KUKA KRL program: MyProgram_164().src

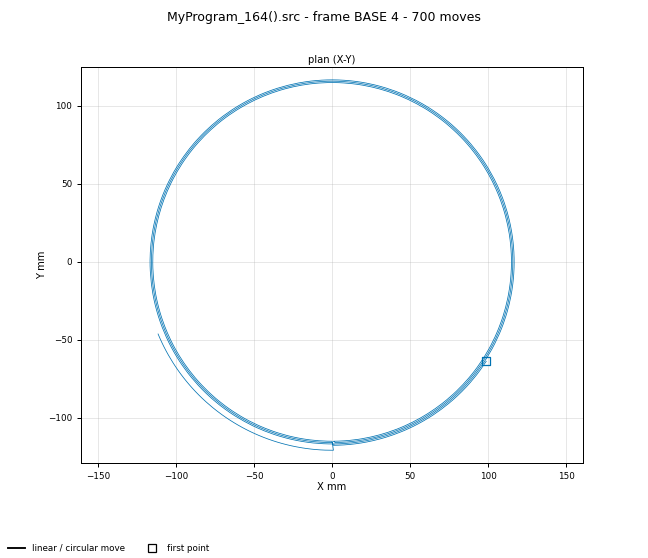
[picture p0: tool path of MyProgram_164().src in frame BASE 4, 700 of 700 moves have a stored position in this frame; points joined in program order, loops and branches not executed]
&ACCESS RVP
&REL 1
&PARAM TEMPLATE = C:\KRC\Roboter\Template\vorgabe
&PARAM EDITMASK = *
DEF MyProgram_164()
; ---- Setting reference (Base) ----
$BASE = BASE_DATA[4]

; --------------------------
; ---- Setting tool (TCP) ----
$TOOL = TOOL_DATA[3]
; --------------------------

$VEL.CP = VEL_APROX_PRINT
Startdeposition()
$VEL.CP = VEL_PRINT
LIN {X 98.7542,Y -63.6993,Z 124,A -36.9555,B 24.954,C -1.5673,E1 25.1338,E2 483.0384} C_DIS
LIN {X 95.0307,Y -69.1319,Z 124,A -40.7241,B 24.956,C -1.5319,E1 25.1276,E2 486.872} C_DIS
LIN {X 92.4043,Y -72.6049,Z 124,A -42.0258,B 24.9541,C -1.565,E1 25.1255,E2 488.0895} C_DIS
LIN {X 88.5317,Y -77.2791,Z 124,A -45.1866,B 24.9551,C -1.5476,E1 25.1198,E2 491.2768} C_DIS
LIN {X 86.1751,Y -79.9009,Z 124,A -47.118,B 24.956,C -1.5331,E1 25.1161,E2 493.234} C_DIS
LIN {X 83.1674,Y -83.0271,Z 124,A -49.5456,B 24.9571,C -1.5131,E1 25.1113,E2 495.6983} C_DIS
LIN {X 80.2255,Y -85.8716,Z 124,A -51.1384,B 24.9563,C -1.5272,E1 25.1081,E2 497.2513} C_DIS
LIN {X 77.3974,Y -88.4284,Z 124,A -52.8872,B 24.9563,C -1.5281,E1 25.1045,E2 498.9912} C_DIS
LIN {X 74.8233,Y -90.6175,Z 124,A -54.4447,B 24.9563,C -1.5286,E1 25.1012,E2 500.5415} C_DIS
LIN {X 69.7732,Y -94.5611,Z 124,A -57.4094,B 24.9562,C -1.5292,E1 25.0947,E2 503.4937} C_DIS
LIN {X 64.9685,Y -97.9241,Z 124,A -60.2141,B 24.9564,C -1.5259,E1 25.0883,E2 506.2966} C_DIS
LIN {X 62.6063,Y -99.4512,Z 124,A -61.8472,B 24.9572,C -1.5109,E1 25.0843,E2 507.9599} C_DIS
LIN {X 58.7888,Y -101.754,Z 124,A -64.5484,B 24.9588,C -1.4824,E1 25.0777,E2 510.7201} C_DIS
LIN {X 55.0039,Y -103.8486,Z 124,A -66.1004,B 24.9576,C -1.5045,E1 25.074,E2 512.2154} C_DIS
LIN {X 51.9264,Y -105.4213,Z 124,A -68.4778,B 24.9595,C -1.4698,E1 25.0679,E2 514.6687} C_DIS
LIN {X 47.367,Y -107.5476,Z 124,A -70.0158,B 24.9574,C -1.5081,E1 25.0642,E2 516.1122} C_DIS
LIN {X 44.6784,Y -108.6919,Z 124,A -71.6622,B 24.9581,C -1.4958,E1 25.0599,E2 517.784} C_DIS
LIN {X 39.1961,Y -110.7866,Z 124,A -74.7628,B 24.9589,C -1.4809,E1 25.0517,E2 520.9132} C_DIS
LIN {X 34.6946,Y -112.2774,Z 124,A -76.7337,B 24.9582,C -1.4937,E1 25.0465,E2 522.85} C_DIS
LIN {X 31.2285,Y -113.2919,Z 124,A -79.3158,B 24.9604,C -1.4543,E1 25.0394,E2 525.5212} C_DIS
LIN {X 26.1754,Y -114.5637,Z 124,A -80.5685,B 24.9572,C -1.5106,E1 25.0363,E2 526.6388} C_DIS
LIN {X 22.2355,Y -115.3928,Z 124,A -82.9862,B 24.9585,C -1.488,E1 25.0296,E2 529.1072} C_DIS
LIN {X 18.6888,Y -116.0221,Z 124,A -84.9192,B 24.959,C -1.4785,E1 25.0242,E2 531.0604} C_DIS
LIN {X 14.9785,Y -116.5572,Z 124,A -86.5895,B 24.9587,C -1.4845,E1 25.0196,E2 532.7153} C_DIS
LIN {X 11.1662,Y -116.9845,Z 124,A -88.5257,B 24.9589,C -1.4804,E1 25.0142,E2 534.6598} C_DIS
LIN {X 7.7029,Y -117.2631,Z 124,A -90.1788,B 24.9589,C -1.4815,E1 25.0096,E2 536.3096} C_DIS
LIN {X 3.8149,Y -117.4539,Z 124,A -92.07,B 24.9589,C -1.4811,E1 25.0043,E2 538.2012} C_DIS
LIN {X 0.8269,Y -117.5118,Z 124,A -92.9024,B 24.9573,C -1.509,E1 25.0022,E2 538.9674} C_DIS
Enddeposition()
LIN {X 0.8269,Y -117.5118,Z 124,A -92.9024,B 24.9573,C -1.509,E1 25.0022,E2 538.9674} C_DIS
Startdeposition()
$VEL.CP = VEL_PRINT
LIN {X 1.3624,Y -116.6412,Z 124,A -92.4871,B 24.9561,C -1.5309,E1 25.0035,E2 538.5001} C_DIS
LIN {X 4.937,Y -116.5432,Z 124,A -90.7988,B 24.9562,C -1.5285,E1 25.0082,E2 536.8181} C_DIS
LIN {X 8.3454,Y -116.3498,Z 124,A -89.0348,B 24.956,C -1.5332,E1 25.0131,E2 535.0436} C_DIS
LIN {X 12.1794,Y -116.0101,Z 124,A -87.2047,B 24.956,C -1.5315,E1 25.0182,E2 533.2187} C_DIS
LIN {X 16.0648,Y -115.5367,Z 124,A -85.3224,B 24.956,C -1.5309,E1 25.0234,E2 531.3393} C_DIS
LIN {X 19.0946,Y -115.0744,Z 124,A -83.8374,B 24.956,C -1.5311,E1 25.0275,E2 529.8554} C_DIS
LIN {X 21.8358,Y -114.5859,Z 124,A -82.4991,B 24.956,C -1.5308,E1 25.0312,E2 528.5191} C_DIS
LIN {X 24.7791,Y -113.9855,Z 124,A -80.9678,B 24.9559,C -1.5347,E1 25.0354,E2 526.9805} C_DIS
LIN {X 33.0953,Y -111.8544,Z 124,A -76.9507,B 24.9562,C -1.5298,E1 25.0462,E2 522.9812} C_DIS
LIN {X 36.0082,Y -110.9509,Z 124,A -75.15,B 24.9552,C -1.5457,E1 25.0511,E2 521.1465} C_DIS
LIN {X 40.8071,Y -109.2778,Z 124,A -72.5586,B 24.9548,C -1.5534,E1 25.0579,E2 518.5422} C_DIS
LIN {X 45.2858,Y -107.4983,Z 124,A -70.3865,B 24.9551,C -1.5477,E1 25.0635,E2 516.3884} C_DIS
LIN {X 47.8668,Y -106.3742,Z 124,A -68.1457,B 24.9526,C -1.5902,E1 25.0694,E2 514.0527} C_DIS
LIN {X 52.9793,Y -103.9226,Z 124,A -66.2695,B 24.9549,C -1.552,E1 25.0739,E2 512.272} C_DIS
LIN {X 58.1058,Y -101.1455,Z 124,A -62.9534,B 24.9533,C -1.5784,E1 25.0821,E2 508.9032} C_DIS
LIN {X 61.3448,Y -99.2159,Z 124,A -61.5325,B 24.9543,C -1.5615,E1 25.0854,E2 507.5266} C_DIS
LIN {X 64.5929,Y -97.1322,Z 124,A -59.0864,B 24.9525,C -1.5914,E1 25.0912,E2 505.0181} C_DIS
LIN {X 68.1356,Y -94.6808,Z 124,A -57.4862,B 24.9537,C -1.5713,E1 25.0947,E2 503.471} C_DIS
LIN {X 73.0483,Y -90.9445,Z 124,A -54.5115,B 24.9535,C -1.5752,E1 25.1013,E2 500.498} C_DIS
LIN {X 75.6279,Y -88.8094,Z 124,A -52.8968,B 24.9534,C -1.5775,E1 25.1047,E2 498.884} C_DIS
LIN {X 78.6353,Y -86.1583,Z 124,A -50.8669,B 24.9529,C -1.585,E1 25.109,E2 496.8446} C_DIS
LIN {X 82.5495,Y -82.4176,Z 124,A -48.2216,B 24.9526,C -1.5908,E1 25.1143,E2 494.1967} C_DIS
LIN {X 84.4942,Y -80.4234,Z 124,A -46.9043,B 24.9526,C -1.5918,E1 25.1168,E2 492.8826} C_DIS
LIN {X 86.8418,Y -77.8794,Z 124,A -45.2097,B 24.9523,C -1.5959,E1 25.12,E2 491.1858} C_DIS
LIN {X 90.3208,Y -73.8178,Z 124,A -42.6097,B 24.9519,C -1.6016,E1 25.1247,E2 488.5843} C_DIS
LIN {X 91.9446,Y -71.7869,Z 124,A -41.019,B 24.9508,C -1.62,E1 25.1275,E2 486.9576} C_DIS
LIN {X 95.3627,Y -67.1797,Z 124,A -38.1108,B 24.9501,C -1.6322,E1 25.1322,E2 484.0347} C_DIS
LIN {X 97.3923,Y -64.1983,Z 124,A -36.8892,B 24.9514,C -1.6108,E1 25.134,E2 482.8696} C_DIS
LIN {X 99.3478,Y -61.132,Z 124,A -35.1139,B 24.9511,C -1.6154,E1 25.1367,E2 481.0925} C_DIS
LIN {X 102.5848,Y -55.5254,Z 124,A -31.853,B 24.9503,C -1.6287,E1 25.1412,E2 477.8173} C_DIS
LIN {X 104.3109,Y -52.2123,Z 124,A -30.2141,B 24.9505,C -1.6248,E1 25.1433,E2 476.1963} C_DIS
LIN {X 107.2037,Y -45.9841,Z 124,A -26.5839,B 24.9491,C -1.6474,E1 25.1475,E2 472.5325} C_DIS
LIN {X 108.4916,Y -42.8522,Z 124,A -25.1108,B 24.9494,C -1.6434,E1 25.149,E2 471.0768} C_DIS
LIN {X 109.6343,Y -39.8375,Z 124,A -22.6264,B 24.9463,C -1.6921,E1 25.1515,E2 468.4916} C_DIS
LIN {X 111.3881,Y -34.6323,Z 124,A -20.7918,B 24.9484,C -1.6587,E1 25.153,E2 466.7461} C_DIS
LIN {X 112.2363,Y -31.7759,Z 124,A -18.7125,B 24.9463,C -1.6932,E1 25.1546,E2 464.5973} C_DIS
LIN {X 113.3809,Y -27.414,Z 124,A -17.6096,B 24.9492,C -1.6466,E1 25.1553,E2 463.6107} C_DIS
LIN {X 114.5448,Y -22.0493,Z 124,A -14.4678,B 24.9473,C -1.6766,E1 25.1572,E2 460.4164} C_DIS
LIN {X 115.1793,Y -18.4619,Z 124,A -12.6055,B 24.9467,C -1.686,E1 25.158,E2 458.5431} C_DIS
LIN {X 115.7491,Y -14.461,Z 124,A -10.6706,B 24.9465,C -1.69,E1 25.1587,E2 456.61} C_DIS
LIN {X 116.1418,Y -10.8535,Z 124,A -8.9547,B 24.9463,C -1.6927,E1 25.1592,E2 454.898} C_DIS
LIN {X 116.3878,Y -7.7827,Z 124,A -7.4105,B 24.9459,C -1.6991,E1 25.1595,E2 453.3478} C_DIS
LIN {X 116.5865,Y -3.7859,Z 124,A -5.5405,B 24.9458,C -1.7009,E1 25.1597,E2 451.4846} C_DIS
LIN {X 116.6446,Y -0.9225,Z 124,A -4.0905,B 24.9454,C -1.7076,E1 25.1597,E2 450.0275} C_DIS
LIN {X 116.6233,Y 2.4022,Z 124,A -2.3642,B 24.9447,C -1.7174,E1 25.1597,E2 448.2884} C_DIS
LIN {X 116.4751,Y 6.3448,Z 124,A -0.61,B 24.9449,C -1.7149,E1 25.1595,E2 446.5506} C_DIS
LIN {X 116.2723,Y 9.3509,Z 124,A 0.8728,B 24.9446,C -1.7198,E1 25.1592,E2 445.0649} C_DIS
LIN {X 115.9636,Y 12.6238,Z 124,A 2.6543,B 24.9437,C -1.733,E1 25.1587,E2 443.2628} C_DIS
LIN {X 115.5191,Y 16.1886,Z 124,A 4.2881,B 24.9437,C -1.7324,E1 25.1581,E2 441.6401} C_DIS
LIN {X 114.9628,Y 19.7618,Z 124,A 6.0877,B 24.9433,C -1.7392,E1 25.1573,E2 439.8351} C_DIS
LIN {X 114.2684,Y 23.44,Z 124,A 7.9174,B 24.943,C -1.7446,E1 25.1563,E2 438.0034} C_DIS
LIN {X 113.3834,Y 27.4035,Z 124,A 9.6005,B 24.9435,C -1.7359,E1 25.1552,E2 436.3505} C_DIS
LIN {X 112.2328,Y 31.788,Z 124,A 12.1154,B 24.9422,C -1.7566,E1 25.1534,E2 433.8013} C_DIS
LIN {X 110.4058,Y 37.6486,Z 124,A 15.0322,B 24.9419,C -1.761,E1 25.1509,E2 430.8906} C_DIS
LIN {X 109.1594,Y 41.1212,Z 124,A 16.9719,B 24.9411,C -1.7725,E1 25.149,E2 428.9346} C_DIS
LIN {X 107.5453,Y 45.1743,Z 124,A 18.989,B 24.9411,C -1.7728,E1 25.1469,E2 426.9279} C_DIS
LIN {X 106.1515,Y 48.3609,Z 124,A 20.7337,B 24.9407,C -1.7795,E1 25.1449,E2 425.177} C_DIS
LIN {X 103.7325,Y 53.3512,Z 124,A 23.4235,B 24.9402,C -1.7856,E1 25.1416,E2 422.4872} C_DIS
LIN {X 100.1461,Y 59.8142,Z 124,A 27.1032,B 24.9394,C -1.7978,E1 25.1365,E2 418.7979} C_DIS
LIN {X 98.2857,Y 62.8224,Z 124,A 28.6878,B 24.9396,C -1.7951,E1 25.1342,E2 417.2275} C_DIS
LIN {X 96.7431,Y 65.1731,Z 124,A 30.6198,B 24.9376,C -1.8249,E1 25.1311,E2 415.2348} C_DIS
LIN {X 94.4395,Y 68.4702,Z 124,A 32.0919,B 24.9389,C -1.806,E1 25.1288,E2 413.8145} C_DIS
LIN {X 92.4871,Y 71.0834,Z 124,A 33.6422,B 24.9388,C -1.8075,E1 25.1261,E2 412.2679} C_DIS
LIN {X 89.196,Y 75.1741,Z 124,A 36.3243,B 24.938,C -1.8185,E1 25.1214,E2 409.5723} C_DIS
LIN {X 86.7479,Y 77.9843,Z 124,A 38.0837,B 24.938,C -1.8194,E1 25.1181,E2 407.8187} C_DIS
LIN {X 84.1411,Y 80.7899,Z 124,A 39.925,B 24.9378,C -1.8217,E1 25.1146,E2 405.9799} C_DIS
LIN {X 81.95,Y 83.0114,Z 124,A 41.4369,B 24.9376,C -1.8241,E1 25.1116,E2 404.4688} C_DIS
LIN {X 79.2815,Y 85.5655,Z 124,A 43.304,B 24.9372,C -1.8303,E1 25.1078,E2 402.5947} C_DIS
LIN {X 76.7637,Y 87.8296,Z 124,A 44.9058,B 24.9372,C -1.8308,E1 25.1045,E2 400.998} C_DIS
LIN {X 74.5063,Y 89.7525,Z 124,A 46.9912,B 24.9349,C -1.863,E1 25.0999,E2 398.8446} C_DIS
LIN {X 70.9944,Y 92.5557,Z 124,A 48.5591,B 24.9367,C -1.8372,E1 25.0965,E2 397.3434} C_DIS
LIN {X 67.7868,Y 94.9297,Z 124,A 50.3301,B 24.9371,C -1.832,E1 25.0926,E2 395.5911} C_DIS
LIN {X 64.3975,Y 97.261,Z 124,A 52.5478,B 24.9362,C -1.8444,E1 25.0874,E2 393.3515} C_DIS
LIN {X 61.3344,Y 99.2224,Z 124,A 54.4921,B 24.9355,C -1.8544,E1 25.0828,E2 391.3897} C_DIS
LIN {X 57.7899,Y 101.327,Z 124,A 56.1965,B 24.9364,C -1.8427,E1 25.0787,E2 389.7182} C_DIS
LIN {X 53.6383,Y 103.5858,Z 124,A 58.7779,B 24.9353,C -1.8577,E1 25.0723,E2 387.1086} C_DIS
LIN {X 47.1433,Y 106.6983,Z 124,A 62.2251,B 24.9353,C -1.8578,E1 25.0636,E2 383.6701} C_DIS
LIN {X 43.3275,Y 108.3047,Z 124,A 64.6027,B 24.9341,C -1.8756,E1 25.0574,E2 381.2557} C_DIS
LIN {X 40.2198,Y 109.4949,Z 124,A 65.8533,B 24.9352,C -1.8597,E1 25.0542,E2 380.0454} C_DIS
LIN {X 36.9579,Y 110.6387,Z 124,A 67.5149,B 24.9352,C -1.8595,E1 25.0498,E2 378.3875} C_DIS
LIN {X 34.4288,Y 111.4512,Z 124,A 69.1235,B 24.9341,C -1.8743,E1 25.0455,E2 376.7468} C_DIS
LIN {X 30.1108,Y 112.6949,Z 124,A 71.3904,B 24.9339,C -1.8785,E1 25.0393,E2 374.4737} C_DIS
LIN {X 26.8729,Y 113.5118,Z 124,A 72.7814,B 24.9346,C -1.8681,E1 25.0356,E2 373.1092} C_DIS
LIN {X 21.9765,Y 114.5588,Z 124,A 75.4902,B 24.9337,C -1.8805,E1 25.0281,E2 370.3744} C_DIS
LIN {X 18.6584,Y 115.1473,Z 124,A 76.9039,B 24.9344,C -1.8702,E1 25.0243,E2 368.9866} C_DIS
LIN {X 15.0241,Y 115.6761,Z 124,A 78.5845,B 24.9348,C -1.8652,E1 25.0197,E2 367.3193} C_DIS
LIN {X 11.6126,Y 116.0695,Z 124,A 80.3473,B 24.9345,C -1.8688,E1 25.0148,E2 365.5491} C_DIS
LIN {X 7.9248,Y 116.3782,Z 124,A 82.1279,B 24.9346,C -1.8672,E1 25.0098,E2 363.7731} C_DIS
LIN {X 3.8833,Y 116.5835,Z 124,A 84.1046,B 24.9346,C -1.8666,E1 25.0043,E2 361.7984} C_DIS
LIN {X 0.3729,Y 116.6476,Z 124,A 85.8948,B 24.9346,C -1.8692,E1 24.9993,E2 360.0022} C_DIS
LIN {X -3.3094,Y 116.6011,Z 124,A 87.5792,B 24.9349,C -1.8633,E1 24.9946,E2 358.3318} C_DIS
LIN {X -6.5798,Y 116.4621,Z 124,A 89.2341,B 24.9349,C -1.8648,E1 24.99,E2 356.6728} C_DIS
LIN {X -10.4984,Y 116.1745,Z 124,A 91.1377,B 24.9349,C -1.8628,E1 24.9847,E2 354.7733} C_DIS
LIN {X -13.5851,Y 115.8539,Z 124,A 92.7068,B 24.9349,C -1.8639,E1 24.9804,E2 353.2005} C_DIS
LIN {X -16.8387,Y 115.4268,Z 124,A 94.5371,B 24.9343,C -1.8724,E1 24.9753,E2 351.3486} C_DIS
LIN {X -21.7106,Y 114.61,Z 124,A 96.7704,B 24.935,C -1.8621,E1 24.9692,E2 349.1374} C_DIS
LIN {X -28.2657,Y 113.1728,Z 124,A 100.1287,B 24.935,C -1.8617,E1 24.96,E2 345.7757} C_DIS
LIN {X -34.9527,Y 111.2887,Z 124,A 103.5513,B 24.9353,C -1.8583,E1 24.9509,E2 342.3555} C_DIS
LIN {X -38.7551,Y 110.0216,Z 124,A 105.4456,B 24.9357,C -1.8527,E1 24.9459,E2 340.4709} C_DIS
LIN {X -43.2758,Y 108.3252,Z 124,A 107.8946,B 24.9357,C -1.8527,E1 24.9395,E2 338.0165} C_DIS
LIN {X -46.5236,Y 106.9685,Z 124,A 109.4387,B 24.9364,C -1.8424,E1 24.9356,E2 336.4935} C_DIS
LIN {X -51.4199,Y 104.7037,Z 124,A 112.2036,B 24.9364,C -1.8431,E1 24.9286,E2 333.72} C_DIS
LIN {X -54.3698,Y 103.2018,Z 124,A 113.8261,B 24.9365,C -1.8403,E1 24.9245,E2 332.0998} C_DIS
LIN {X -57.27,Y 101.6221,Z 124,A 115.4265,B 24.9368,C -1.8365,E1 24.9206,E2 330.5038} C_DIS
LIN {X -60.9655,Y 99.449,Z 124,A 118.0379,B 24.9356,C -1.8541,E1 24.9143,E2 327.8426} C_DIS
LIN {X -64.0825,Y 97.4687,Z 124,A 119.3881,B 24.9372,C -1.8309,E1 24.9112,E2 326.5431} C_DIS
LIN {X -69.7578,Y 93.4916,Z 124,A 123.3224,B 24.9361,C -1.8462,E1 24.9022,E2 322.5585} C_DIS
LIN {X -72.9301,Y 91.0403,Z 124,A 124.8934,B 24.9376,C -1.8251,E1 24.8989,E2 321.0321} C_DIS
LIN {X -77.1018,Y 87.5343,Z 124,A 127.5382,B 24.9381,C -1.8177,E1 24.8933,E2 318.3945} C_DIS
LIN {X -79.6573,Y 85.2146,Z 124,A 129.1643,B 24.9385,C -1.8108,E1 24.89,E2 316.7782} C_DIS
LIN {X -81.473,Y 83.4824,Z 124,A 130.4942,B 24.9385,C -1.8119,E1 24.8873,E2 315.4402} C_DIS
LIN {X -83.8363,Y 81.1062,Z 124,A 132.2471,B 24.9385,C -1.8123,E1 24.8838,E2 313.6788} C_DIS
LIN {X -86.6399,Y 78.1049,Z 124,A 134.1116,B 24.9392,C -1.8008,E1 24.8804,E2 311.8335} C_DIS
LIN {X -88.5148,Y 75.9738,Z 124,A 135.6705,B 24.939,C -1.8041,E1 24.8775,E2 310.2597} C_DIS
LIN {X -91.269,Y 72.6417,Z 124,A 137.668,B 24.9397,C -1.7932,E1 24.874,E2 308.2789} C_DIS
LIN {X -95.079,Y 67.5775,Z 124,A 141.0042,B 24.9397,C -1.7939,E1 24.8685,E2 304.9249} C_DIS
LIN {X -98.2141,Y 62.9341,Z 124,A 143.5663,B 24.9407,C -1.7783,E1 24.8645,E2 302.3872} C_DIS
LIN {X -99.5689,Y 60.7682,Z 124,A 145.2412,B 24.9398,C -1.792,E1 24.8621,E2 300.6708} C_DIS
LIN {X -101.4314,Y 57.6082,Z 124,A 147.1001,B 24.94,C -1.7891,E1 24.8595,E2 298.8092} C_DIS
LIN {X -103.2054,Y 54.363,Z 124,A 148.3584,B 24.9419,C -1.7606,E1 24.8579,E2 297.6121} C_DIS
LIN {X -104.4149,Y 52.0025,Z 124,A 149.7102,B 24.942,C -1.7587,E1 24.8562,E2 296.2576} C_DIS
LIN {X -105.6333,Y 49.481,Z 124,A 151.1826,B 24.942,C -1.7586,E1 24.8544,E2 294.7776} C_DIS
LIN {X -107.0948,Y 46.2339,Z 124,A 152.9845,B 24.9422,C -1.7554,E1 24.8524,E2 292.9734} C_DIS
LIN {X -108.5301,Y 42.7541,Z 124,A 154.8745,B 24.9425,C -1.7514,E1 24.8504,E2 291.0824} C_DIS
LIN {X -110.0165,Y 38.7696,Z 124,A 156.8052,B 24.9434,C -1.7383,E1 24.8486,E2 289.172} C_DIS
LIN {X -110.9839,Y 35.9064,Z 124,A 158.3608,B 24.9434,C -1.7365,E1 24.8472,E2 287.6116} C_DIS
LIN {X -112.0389,Y 32.4724,Z 124,A 160.4445,B 24.943,C -1.744,E1 24.8456,E2 285.4981} C_DIS
LIN {X -113.2143,Y 28.0967,Z 124,A 162.2202,B 24.9447,C -1.7184,E1 24.8444,E2 283.7731} C_DIS
LIN {X -114.1826,Y 23.8578,Z 124,A 164.4125,B 24.945,C -1.7138,E1 24.843,E2 281.5788} C_DIS
LIN {X -114.6949,Y 21.2641,Z 124,A 165.9136,B 24.9447,C -1.7179,E1 24.8422,E2 280.0591} C_DIS
LIN {X -115.3693,Y 17.2328,Z 124,A 168.0274,B 24.9448,C -1.7158,E1 24.8413,E2 277.9379} C_DIS
LIN {X -116.0541,Y 11.7593,Z 124,A 170.6852,B 24.9455,C -1.7048,E1 24.8405,E2 275.2902} C_DIS
LIN {X -116.4878,Y 6.1072,Z 124,A 173.6084,B 24.9457,C -1.7014,E1 24.8399,E2 272.3575} C_DIS
LIN {X -116.6433,Y 1.1077,Z 124,A 175.8997,B 24.9467,C -1.6866,E1 24.8398,E2 270.0878} C_DIS
LIN {X -116.6229,Y -2.4209,Z 124,A 177.5955,B 24.9471,C -1.6794,E1 24.8398,E2 268.3989} C_DIS
LIN {X -116.498,Y -5.9283,Z 124,A 179.4939,B 24.9471,C -1.681,E1 24.8401,E2 266.4853} C_DIS
LIN {X -115.7697,Y -14.3023,Z 124,A -176.2617,B 24.9476,C -1.6724,E1 24.8413,E2 262.236} C_DIS
LIN {X -114.8264,Y -20.5328,Z 124,A -172.8352,B 24.9473,C -1.6763,E1 24.8428,E2 258.7797} C_DIS
LIN {X -114.039,Y -24.5339,Z 124,A -171.3242,B 24.949,C -1.6496,E1 24.8437,E2 257.3235} C_DIS
LIN {X -113.287,Y -27.7986,Z 124,A -169.2783,B 24.9483,C -1.6611,E1 24.845,E2 255.2383} C_DIS
LIN {X -112.3749,Y -31.2866,Z 124,A -167.8442,B 24.9495,C -1.6416,E1 24.8461,E2 253.8423} C_DIS
LIN {X -111.3302,Y -34.8191,Z 124,A -166.0795,B 24.95,C -1.6342,E1 24.8475,E2 252.085} C_DIS
LIN {X -110.1425,Y -38.4105,Z 124,A -164.1882,B 24.9502,C -1.63,E1 24.8492,E2 250.193} C_DIS
LIN {X -108.833,Y -41.983,Z 124,A -162.2156,B 24.9502,C -1.6287,E1 24.8511,E2 248.2124} C_DIS
LIN {X -106.2298,Y -48.1873,Z 124,A -158.9883,B 24.9511,C -1.6159,E1 24.8547,E2 244.9978} C_DIS
LIN {X -104.7752,Y -51.2758,Z 124,A -157.21,B 24.9511,C -1.6153,E1 24.8569,E2 243.2112} C_DIS
LIN {X -103.1018,Y -54.5597,Z 124,A -155.5677,B 24.9518,C -1.6033,E1 24.8589,E2 241.5888} C_DIS
LIN {X -101.3249,Y -57.7935,Z 124,A -153.6752,B 24.9519,C -1.6017,E1 24.8615,E2 239.6903} C_DIS
LIN {X -99.7723,Y -60.4336,Z 124,A -151.8165,B 24.9513,C -1.6125,E1 24.8643,E2 237.7961} C_DIS
LIN {X -98.0488,Y -63.1915,Z 124,A -150.5899,B 24.9525,C -1.5927,E1 24.8661,E2 236.6105} C_DIS
LIN {X -96.1967,Y -65.9801,Z 124,A -148.8284,B 24.9525,C -1.5934,E1 24.8688,E2 234.8387} C_DIS
LIN {X -94.1441,Y -68.8737,Z 124,A -147.1468,B 24.9528,C -1.5865,E1 24.8716,E2 233.1653} C_DIS
LIN {X -92.5609,Y -70.9876,Z 124,A -145.3656,B 24.9518,C -1.6038,E1 24.8747,E2 231.3344} C_DIS
LIN {X -90.116,Y -74.0689,Z 124,A -144.0026,B 24.9535,C -1.575,E1 24.877,E2 230.0336} C_DIS
LIN {X -85.6839,Y -79.1525,Z 124,A -140.4608,B 24.9534,C -1.5771,E1 24.8836,E2 226.471} C_DIS
LIN {X -83.006,Y -81.9554,Z 124,A -138.6761,B 24.9539,C -1.5679,E1 24.887,E2 224.7006} C_DIS
LIN {X -81.0293,Y -83.9104,Z 124,A -137.2764,B 24.954,C -1.5664,E1 24.8898,E2 223.2984} C_DIS
LIN {X -78.1281,Y -86.6191,Z 124,A -135.516,B 24.9547,C -1.5544,E1 24.8934,E2 221.5595} C_DIS
LIN {X -75.9544,Y -88.53,Z 124,A -133.151,B 24.9525,C -1.5922,E1 24.8986,E2 219.0954} C_DIS
LIN {X -71.9938,Y -91.7811,Z 124,A -131.2622,B 24.9544,C -1.5603,E1 24.9026,E2 217.2754} C_DIS
LIN {X -68.7307,Y -94.2488,Z 124,A -129.2623,B 24.9546,C -1.5564,E1 24.9071,E2 215.2778} C_DIS
LIN {X -65.5885,Y -96.4618,Z 124,A -127.425,B 24.9549,C -1.551,E1 24.9113,E2 213.4469} C_DIS
LIN {X -62.3223,Y -98.6053,Z 124,A -125.4267,B 24.9549,C -1.5514,E1 24.916,E2 211.4413} C_DIS
LIN {X -56.3389,Y -102.142,Z 124,A -122.2059,B 24.9557,C -1.5381,E1 24.9237,E2 208.2425} C_DIS
LIN {X -50.9398,Y -104.9383,Z 124,A -119.0798,B 24.9555,C -1.5403,E1 24.9315,E2 205.1027} C_DIS
LIN {X -47.9027,Y -106.358,Z 124,A -117.4982,B 24.9558,C -1.5356,E1 24.9355,E2 203.5284} C_DIS
LIN {X -43.039,Y -108.4182,Z 124,A -114.8225,B 24.9558,C -1.5365,E1 24.9424,E2 200.8447} C_DIS
LIN {X -39.7365,Y -109.6712,Z 124,A -113.1495,B 24.956,C -1.5321,E1 24.9468,E2 199.1785} C_DIS
LIN {X -37.2124,Y -110.5528,Z 124,A -111.5694,B 24.9554,C -1.5428,E1 24.9511,E2 197.5699} C_DIS
LIN {X -33.5458,Y -111.7207,Z 124,A -109.5834,B 24.9552,C -1.5457,E1 24.9564,E2 195.5738} C_DIS
LIN {X -29.0685,Y -112.9678,Z 124,A -107.6872,B 24.9563,C -1.5271,E1 24.9614,E2 193.7188} C_DIS
LIN {X -26.3497,Y -113.6327,Z 124,A -106.2072,B 24.9561,C -1.5311,E1 24.9654,E2 192.2275} C_DIS
LIN {X -22.5124,Y -114.4557,Z 124,A -104.2673,B 24.9561,C -1.5308,E1 24.9708,E2 190.286} C_DIS
LIN {X -19.1502,Y -115.0651,Z 124,A -102.6503,B 24.9563,C -1.5275,E1 24.9752,E2 188.6753} C_DIS
LIN {X -15.2619,Y -115.6453,Z 124,A -100.8004,B 24.9565,C -1.5234,E1 24.9803,E2 186.8336} C_DIS
LIN {X -12.0498,Y -116.0237,Z 124,A -99.1028,B 24.9563,C -1.5281,E1 24.985,E2 185.1238} C_DIS
LIN {X -8.1648,Y -116.362,Z 124,A -97.2841,B 24.9565,C -1.5237,E1 24.9901,E2 183.3147} C_DIS
LIN {X -5.6175,Y -116.5133,Z 124,A -95.9012,B 24.9562,C -1.5296,E1 24.994,E2 181.9175} C_DIS
LIN {X -2.1692,Y -116.6276,Z 124,A -94.2855,B 24.9564,C -1.5263,E1 24.9984,E2 180.3094} C_DIS
LIN {X 0.8245,Y -116.6427,Z 124,A -93.3941,B 24.9578,C -1.5006,E1 25.0008,E2 179.4789} C_DIS
Enddeposition()
LIN {X 0.8245,Y -116.6427,Z 124,A -93.3941,B 24.9578,C -1.5006,E1 25.0008,E2 179.4789} C_DIS
Startdeposition()
$VEL.CP = VEL_PRINT
LIN {X -0.0422,Y -115.7818,Z 124,A -94.1118,B 24.9577,C -1.5029,E1 24.9988,E2 180.1911} C_DIS
LIN {X -3.596,Y -115.724,Z 124,A -95.6773,B 24.9572,C -1.5112,E1 24.9945,E2 181.7372} C_DIS
LIN {X -6.6918,Y -115.5867,Z 124,A -97.2377,B 24.9572,C -1.5099,E1 24.9901,E2 183.301} C_DIS
LIN {X -10.2839,Y -115.3228,Z 124,A -99.0208,B 24.9572,C -1.5099,E1 24.9851,E2 185.0848} C_DIS
LIN {X -12.8754,Y -115.0632,Z 124,A -100.4846,B 24.9577,C -1.5024,E1 24.981,E2 186.5674} C_DIS
LIN {X -16.5458,Y -114.5918,Z 124,A -102.2637,B 24.9576,C -1.5051,E1 24.9761,E2 188.3415} C_DIS
LIN {X -19.9681,Y -114.0462,Z 124,A -103.9919,B 24.9576,C -1.5051,E1 24.9713,E2 190.0715} C_DIS
LIN {X -22.9478,Y -113.4834,Z 124,A -105.2898,B 24.957,C -1.5144,E1 24.9678,E2 191.3484} C_DIS
LIN {X -25.2419,Y -112.9963,Z 124,A -106.8395,B 24.958,C -1.4981,E1 24.9635,E2 192.9389} C_DIS
LIN {X -29.5057,Y -111.9592,Z 124,A -108.727,B 24.9572,C -1.5116,E1 24.9585,E2 194.797} C_DIS
LIN {X -32.3563,Y -111.1683,Z 124,A -110.3907,B 24.9576,C -1.504,E1 24.954,E2 196.4815} C_DIS
LIN {X -36.0487,Y -110.0257,Z 124,A -112.272,B 24.9575,C -1.5068,E1 24.949,E2 198.3594} C_DIS
LIN {X -39.2828,Y -108.9128,Z 124,A -113.6426,B 24.9566,C -1.5221,E1 24.9454,E2 199.6963} C_DIS
LIN {X -41.3773,Y -108.1344,Z 124,A -114.9491,B 24.957,C -1.5145,E1 24.942,E2 201.0236} C_DIS
LIN {X -45.0569,Y -106.653,Z 124,A -116.9742,B 24.957,C -1.5139,E1 24.9367,E2 203.0547} C_DIS
LIN {X -48.7207,Y -105.0299,Z 124,A -118.8384,B 24.9566,C -1.5212,E1 24.932,E2 204.9061} C_DIS
LIN {X -52.5733,Y -103.1554,Z 124,A -121.0937,B 24.9568,C -1.5181,E1 24.9263,E2 207.1747} C_DIS
LIN {X -56.0252,Y -101.3232,Z 124,A -122.9632,B 24.9565,C -1.5234,E1 24.9218,E2 209.0369} C_DIS
LIN {X -59.6868,Y -99.2105,Z 124,A -124.9633,B 24.9561,C -1.5304,E1 24.917,E2 211.0265} C_DIS
LIN {X -62.4196,Y -97.513,Z 124,A -126.6449,B 24.9561,C -1.5291,E1 24.913,E2 212.7165} C_DIS
LIN {X -65.318,Y -95.5969,Z 124,A -128.5187,B 24.9564,C -1.5254,E1 24.9086,E2 214.6054} C_DIS
LIN {X -68.5163,Y -93.3301,Z 124,A -130.4248,B 24.9561,C -1.5301,E1 24.9043,E2 216.5068} C_DIS
LIN {X -71.972,Y -90.6921,Z 124,A -133.4816,B 24.958,C -1.4966,E1 24.8974,E2 219.6546} C_DIS
LIN {X -76.6836,Y -86.7472,Z 124,A -135.4828,B 24.9552,C -1.5455,E1 24.8934,E2 221.5474} C_DIS
LIN {X -79.6326,Y -84.0464,Z 124,A -137.5238,B 24.9552,C -1.547,E1 24.8892,E2 223.5931} C_DIS
LIN {X -82.15,Y -81.587,Z 124,A -139.299,B 24.955,C -1.5493,E1 24.8857,E2 225.3703} C_DIS
LIN {X -84.9958,Y -78.6187,Z 124,A -141.8744,B 24.9561,C -1.5316,E1 24.8807,E2 227.9991} C_DIS
LIN {X -87.7517,Y -75.5311,Z 124,A -143.2769,B 24.9542,C -1.5628,E1 24.8782,E2 229.3336} C_DIS
LIN {X -89.6499,Y -73.2672,Z 124,A -145.0165,B 24.9547,C -1.5548,E1 24.8751,E2 231.1002} C_DIS
LIN {X -92.1975,Y -70.0352,Z 124,A -146.9588,B 24.9542,C -1.5637,E1 24.8718,E2 233.0307} C_DIS
LIN {X -93.9354,Y -67.686,Z 124,A -148.2208,B 24.9535,C -1.5749,E1 24.8697,E2 234.2722} C_DIS
LIN {X -95.2585,Y -65.8095,Z 124,A -149.6237,B 24.954,C -1.5668,E1 24.8675,E2 235.7011} C_DIS
LIN {X -97.1533,Y -62.98,Z 124,A -151.0497,B 24.9531,C -1.5818,E1 24.8653,E2 237.0986} C_DIS
LIN {X -98.2787,Y -61.2069,Z 124,A -152.3631,B 24.9536,C -1.5734,E1 24.8633,E2 238.4389} C_DIS
LIN {X -100.3558,Y -57.738,Z 124,A -154.3082,B 24.9532,C -1.581,E1 24.8606,E2 240.3758} C_DIS
LIN {X -102.4039,Y -54.0224,Z 124,A -156.2743,B 24.9525,C -1.5923,E1 24.858,E2 242.3254} C_DIS
LIN {X -103.7001,Y -51.4904,Z 124,A -157.7403,B 24.9525,C -1.5938,E1 24.8561,E2 243.7956} C_DIS
LIN {X -105.233,Y -48.2845,Z 124,A -159.7043,B 24.9526,C -1.5905,E1 24.8538,E2 245.7782} C_DIS
LIN {X -106.4373,Y -45.5687,Z 124,A -161.292,B 24.9526,C -1.59,E1 24.852,E2 247.3759} C_DIS
LIN {X -108.2244,Y -41.1397,Z 124,A -163.3931,B 24.9516,C -1.6076,E1 24.8499,E2 249.4468} C_DIS
LIN {X -109.4716,Y -37.7012,Z 124,A -165.1706,B 24.9512,C -1.6143,E1 24.8483,E2 251.2184} C_DIS
LIN {X -110.3851,Y -34.9364,Z 124,A -166.7501,B 24.9512,C -1.6131,E1 24.8469,E2 252.8099} C_DIS
LIN {X -111.5631,Y -30.9683,Z 124,A -168.8202,B 24.9509,C -1.6185,E1 24.8453,E2 254.879} C_DIS
LIN {X -112.5089,Y -27.3264,Z 124,A -170.632,B 24.9504,C -1.6264,E1 24.8441,E2 256.6827} C_DIS
LIN {X -113.3734,Y -23.4839,Z 124,A -172.648,B 24.9502,C -1.6298,E1 24.8429,E2 258.7025} C_DIS
LIN {X -114.4548,Y -17.4674,Z 124,A -175.68,B 24.9497,C -1.6391,E1 24.8414,E2 261.7302} C_DIS
LIN {X -114.9715,Y -13.6583,Z 124,A -177.8676,B 24.95,C -1.6338,E1 24.8407,E2 263.9436} C_DIS
LIN {X -115.5236,Y -7.6987,Z 124,A 179.9064,B 24.9476,C -1.6729,E1 24.8402,E2 266.0897} C_DIS
LIN {X -115.735,Y -3.2375,Z 124,A 177.1302,B 24.9485,C -1.6573,E1 24.8398,E2 268.9198} C_DIS
LIN {X -115.778,Y 0.7173,Z 124,A 174.8092,B 24.949,C -1.6491,E1 24.8398,E2 271.2742} C_DIS
LIN {X -115.6929,Y 4.5094,Z 124,A 172.4654,B 24.9498,C -1.6369,E1 24.8401,E2 273.6614} C_DIS
LIN {X -115.3256,Y 10.253,Z 124,A 170.1633,B 24.9479,C -1.6677,E1 24.8406,E2 275.9038} C_DIS
LIN {X -114.9957,Y 13.4524,Z 124,A 168.8931,B 24.9467,C -1.6857,E1 24.841,E2 277.1387} C_DIS
LIN {X -114.4868,Y 17.2605,Z 124,A 166.91,B 24.9466,C -1.6886,E1 24.8418,E2 279.1267} C_DIS
LIN {X -113.8218,Y 21.2142,Z 124,A 164.8586,B 24.9463,C -1.6923,E1 24.8428,E2 281.1814} C_DIS
LIN {X -113.0172,Y 25.1457,Z 124,A 162.9566,B 24.9457,C -1.7021,E1 24.8439,E2 283.0713} C_DIS
LIN {X -112.3287,Y 28.0651,Z 124,A 161.3737,B 24.9457,C -1.7029,E1 24.845,E2 284.6615} C_DIS
LIN {X -111.3942,Y 31.5644,Z 124,A 159.8261,B 24.9447,C -1.7185,E1 24.8461,E2 286.181} C_DIS
LIN {X -110.7251,Y 33.8399,Z 124,A 158.6605,B 24.9444,C -1.7225,E1 24.847,E2 287.3437} C_DIS
LIN {X -109.94,Y 36.3133,Z 124,A 157.07,B 24.9449,C -1.7143,E1 24.8484,E2 288.9629} C_DIS
LIN {X -108.5569,Y 40.2587,Z 124,A 154.9971,B 24.9445,C -1.7206,E1 24.8504,E2 291.0324} C_DIS
LIN {X -107.0554,Y 44.0948,Z 124,A 153.0599,B 24.9438,C -1.731,E1 24.8524,E2 292.9558} C_DIS
LIN {X -105.8796,Y 46.8495,Z 124,A 151.4353,B 24.9439,C -1.7298,E1 24.8542,E2 294.5921} C_DIS
LIN {X -104.04,Y 50.8047,Z 124,A 149.5002,B 24.9429,C -1.7453,E1 24.8565,E2 296.5008} C_DIS
LIN {X -102.5803,Y 53.6875,Z 124,A 148.0666,B 24.9422,C -1.7568,E1 24.8583,E2 297.9147} C_DIS
LIN {X -101.3849,Y 55.9132,Z 124,A 146.4577,B 24.9429,C -1.746,E1 24.8605,E2 299.5577} C_DIS
LIN {X -99.594,Y 59.0425,Z 124,A 144.769,B 24.9423,C -1.7551,E1 24.8628,E2 301.2336} C_DIS
LIN {X -97.7522,Y 62.047,Z 124,A 142.9477,B 24.9421,C -1.7569,E1 24.8655,E2 303.0598} C_DIS
LIN {X -94.9457,Y 66.2595,Z 124,A 140.1666,B 24.9424,C -1.7529,E1 24.87,E2 305.8643} C_DIS
LIN {X -93.0698,Y 68.8718,Z 124,A 138.5204,B 24.9423,C -1.755,E1 24.8727,E2 307.5133} C_DIS
LIN {X -91.088,Y 71.4711,Z 124,A 137.3703,B 24.9407,C -1.7782,E1 24.8746,E2 308.6136} C_DIS
LIN {X -88.1939,Y 75.0121,Z 124,A 134.9223,B 24.9408,C -1.7767,E1 24.879,E2 311.0765} C_DIS
LIN {X -85.6311,Y 77.9263,Z 124,A 133.0489,B 24.9404,C -1.7835,E1 24.8824,E2 312.9421} C_DIS
LIN {X -82.8688,Y 80.8594,Z 124,A 130.9473,B 24.9404,C -1.7841,E1 24.8865,E2 315.0515} C_DIS
LIN {X -80.3671,Y 83.3433,Z 124,A 129.2348,B 24.94,C -1.7897,E1 24.8899,E2 316.7578} C_DIS
LIN {X -77.1497,Y 86.3302,Z 124,A 127.044,B 24.9397,C -1.794,E1 24.8944,E2 318.9471} C_DIS
LIN {X -73.7303,Y 89.2688,Z 124,A 124.9561,B 24.9389,C -1.8049,E1 24.8988,E2 321.0172} C_DIS
LIN {X -69.1099,Y 92.8929,Z 124,A 121.7872,B 24.9392,C -1.8003,E1 24.9059,E2 324.2085} C_DIS
LIN {X -65.8832,Y 95.2073,Z 124,A 120.0016,B 24.9385,C -1.8117,E1 24.9099,E2 325.9732} C_DIS
LIN {X -63.4856,Y 96.8227,Z 124,A 118.3091,B 24.939,C -1.8038,E1 24.9139,E2 327.6902} C_DIS
LIN {X -59.4627,Y 99.3457,Z 124,A 116.2735,B 24.9378,C -1.8211,E1 24.9187,E2 329.6909} C_DIS
LIN {X -56.5911,Y 101.0072,Z 124,A 114.661,B 24.9376,C -1.8253,E1 24.9226,E2 331.2982} C_DIS
LIN {X -53.5762,Y 102.6389,Z 124,A 112.7081,B 24.9381,C -1.8175,E1 24.9274,E2 333.275} C_DIS
LIN {X -49.6654,Y 104.5878,Z 124,A 110.5273,B 24.9379,C -1.8202,E1 24.9329,E2 335.4551} C_DIS
LIN {X -46.5438,Y 106.0129,Z 124,A 108.9385,B 24.9374,C -1.8273,E1 24.9369,E2 337.0307} C_DIS
LIN {X -43.543,Y 107.2799,Z 124,A 107.3412,B 24.9372,C -1.8302,E1 24.9411,E2 338.6248} C_DIS
LIN {X -39.9798,Y 108.6586,Z 124,A 105.657,B 24.9364,C -1.8414,E1 24.9454,E2 340.2859} C_DIS
LIN {X -37.116,Y 109.6694,Z 124,A 104.1445,B 24.9364,C -1.8429,E1 24.9494,E2 341.7978} C_DIS
LIN {X -34.97,Y 110.3747,Z 124,A 102.8769,B 24.9367,C -1.8379,E1 24.9528,E2 343.0797} C_DIS
LIN {X -31.6836,Y 111.3604,Z 124,A 101.1023,B 24.9367,C -1.8366,E1 24.9576,E2 344.8603} C_DIS
LIN {X -23.4956,Y 113.371,Z 124,A 97.1656,B 24.9358,C -1.8505,E1 24.9682,E2 348.7693} C_DIS
LIN {X -17.4562,Y 114.4566,Z 124,A 93.8607,B 24.9364,C -1.8413,E1 24.9773,E2 352.0993} C_DIS
LIN {X -14.0448,Y 114.9263,Z 124,A 92.1066,B 24.9365,C -1.8402,E1 24.9822,E2 353.8573} C_DIS
LIN {X -10.4865,Y 115.3041,Z 124,A 90.4061,B 24.9363,C -1.8441,E1 24.9869,E2 355.5494} C_DIS
LIN {X -6.3497,Y 115.6056,Z 124,A 88.3243,B 24.9363,C -1.8437,E1 24.9927,E2 357.633} C_DIS
LIN {X -2.8414,Y 115.7471,Z 124,A 86.4963,B 24.9365,C -1.8403,E1 24.9978,E2 359.4693} C_DIS
LIN {X 0.6566,Y 115.778,Z 124,A 84.8925,B 24.9361,C -1.8462,E1 25.0023,E2 361.0591} C_DIS
LIN {X 3.9273,Y 115.7138,Z 124,A 83.1463,B 24.9365,C -1.8408,E1 25.0072,E2 362.8176} C_DIS
LIN {X 7.8542,Y 115.5131,Z 124,A 81.3363,B 24.9361,C -1.8467,E1 25.0122,E2 364.6129} C_DIS
LIN {X 11.0337,Y 115.2536,Z 124,A 79.635,B 24.9365,C -1.8413,E1 25.0169,E2 366.3262} C_DIS
LIN {X 14.8254,Y 114.8267,Z 124,A 77.8648,B 24.9361,C -1.846,E1 25.0218,E2 368.0838} C_DIS
LIN {X 17.9891,Y 114.3742,Z 124,A 75.2875,B 24.9391,C -1.8025,E1 25.0292,E2 370.7618} C_DIS
LIN {X 23.9763,Y 113.2705,Z 124,A 73.2074,B 24.9364,C -1.8415,E1 25.0346,E2 372.7469} C_DIS
LIN {X 27.2588,Y 112.5254,Z 124,A 71.506,B 24.9366,C -1.839,E1 25.0393,E2 374.4517} C_DIS
LIN {X 31.5514,Y 111.3978,Z 124,A 69.403,B 24.9364,C -1.8417,E1 25.0449,E2 376.5451} C_DIS
LIN {X 35.3597,Y 110.2486,Z 124,A 67.5579,B 24.9362,C -1.8456,E1 25.0498,E2 378.3776} C_DIS
LIN {X 37.6442,Y 109.4913,Z 124,A 66.3151,B 24.9364,C -1.8422,E1 25.0531,E2 379.6259} C_DIS
LIN {X 40.7476,Y 108.3729,Z 124,A 64.6031,B 24.9367,C -1.8372,E1 25.0576,E2 381.3463} C_DIS
LIN {X 44.3301,Y 106.9592,Z 124,A 62.601,B 24.9372,C -1.8309,E1 25.0628,E2 383.3586} C_DIS
LIN {X 50.5956,Y 104.1408,Z 124,A 59.3141,B 24.9371,C -1.8319,E1 25.0711,E2 386.6348} C_DIS
LIN {X 53.8429,Y 102.4984,Z 124,A 57.3009,B 24.9379,C -1.8201,E1 25.0762,E2 388.6704} C_DIS
LIN {X 57.2162,Y 100.6557,Z 124,A 55.7737,B 24.9369,C -1.8342,E1 25.0798,E2 390.1599} C_DIS
LIN {X 60.0481,Y 98.9909,Z 124,A 54.0467,B 24.9374,C -1.8272,E1 25.084,E2 391.898} C_DIS
LIN {X 62.7211,Y 97.3195,Z 124,A 52.6375,B 24.9371,C -1.8316,E1 25.0873,E2 393.2924} C_DIS
LIN {X 64.912,Y 95.8718,Z 124,A 51.1558,B 24.9378,C -1.8212,E1 25.0908,E2 394.7936} C_DIS
LIN {X 68.1324,Y 93.6112,Z 124,A 49.1866,B 24.9381,C -1.8168,E1 25.0952,E2 396.7663} C_DIS
LIN {X 71.1106,Y 91.3704,Z 124,A 47.3616,B 24.9383,C -1.8143,E1 25.0993,E2 398.5906} C_DIS
LIN {X 74.6377,Y 88.5128,Z 124,A 45.0833,B 24.9387,C -1.8086,E1 25.1042,E2 400.8738} C_DIS
LIN {X 77.1173,Y 86.3592,Z 124,A 43.5259,B 24.9387,C -1.8084,E1 25.1075,E2 402.4253} C_DIS
LIN {X 79.7004,Y 83.9826,Z 124,A 41.8064,B 24.9389,C -1.8056,E1 25.111,E2 404.1445} C_DIS
LIN {X 82.2787,Y 81.4567,Z 124,A 40.0782,B 24.9389,C -1.8044,E1 25.1144,E2 405.8682} C_DIS
LIN {X 84.4874,Y 79.1637,Z 124,A 38.4774,B 24.9393,C -1.7998,E1 25.1175,E2 407.473} C_DIS
LIN {X 86.9895,Y 76.4062,Z 124,A 36.6333,B 24.9396,C -1.7955,E1 25.1209,E2 409.3191} C_DIS
LIN {X 89.6511,Y 73.2658,Z 124,A 34.5321,B 24.9401,C -1.7877,E1 25.1247,E2 411.4291} C_DIS
LIN {X 92.0133,Y 70.2763,Z 124,A 32.7761,B 24.9401,C -1.789,E1 25.1277,E2 413.1736} C_DIS
LIN {X 94.0844,Y 67.4772,Z 124,A 31.2589,B 24.9397,C -1.7942,E1 25.1302,E2 414.6711} C_DIS
LIN {X 95.786,Y 65.0387,Z 124,A 29.7129,B 24.9401,C -1.787,E1 25.1326,E2 416.2266} C_DIS
LIN {X 97.0846,Y 63.087,Z 124,A 28.2856,B 24.9412,C -1.7716,E1 25.1349,E2 417.6832} C_DIS
LIN {X 99.3371,Y 59.4772,Z 124,A 25.8273,B 24.9426,C -1.7496,E1 25.1385,E2 420.1807} C_DIS
LIN {X 101.1826,Y 56.2769,Z 124,A 24.5198,B 24.9414,C -1.7687,E1 25.1402,E2 421.4364} C_DIS
LIN {X 102.8866,Y 53.0992,Z 124,A 22.3536,B 24.9429,C -1.746,E1 25.1431,E2 423.6446} C_DIS
LIN {X 104.3183,Y 50.2262,Z 124,A 21.2426,B 24.9417,C -1.7637,E1 25.1444,E2 424.708} C_DIS
LIN {X 105.3394,Y 48.0505,Z 124,A 20.086,B 24.9418,C -1.7618,E1 25.1457,E2 425.8629} C_DIS
LIN {X 106.6045,Y 45.1719,Z 124,A 18.3889,B 24.9426,C -1.7507,E1 25.1476,E2 427.5769} C_DIS
LIN {X 107.8585,Y 42.0901,Z 124,A 16.874,B 24.9425,C -1.752,E1 25.1492,E2 429.0804} C_DIS
LIN {X 109.0169,Y 38.9973,Z 124,A 15.2032,B 24.9429,C -1.7454,E1 25.1508,E2 430.7575} C_DIS
LIN {X 109.7655,Y 36.8312,Z 124,A 14.013,B 24.9433,C -1.7393,E1 25.1519,E2 431.9551} C_DIS
LIN {X 111.1101,Y 32.5526,Z 124,A 11.3769,B 24.945,C -1.7131,E1 25.154,E2 434.6381} C_DIS
LIN {X 112.0677,Y 29.0838,Z 124,A 9.8932,B 24.9445,C -1.7214,E1 25.1551,E2 436.0936} C_DIS
LIN {X 113.1554,Y 24.5124,Z 124,A 7.666,B 24.9446,C -1.7187,E1 25.1564,E2 438.3142} C_DIS
LIN {X 113.8579,Y 21.0151,Z 124,A 6.115,B 24.9443,C -1.7232,E1 25.1573,E2 439.8456} C_DIS
LIN {X 114.3981,Y 17.8341,Z 124,A 4.3975,B 24.945,C -1.7125,E1 25.1581,E2 441.5783} C_DIS
LIN {X 114.8695,Y 14.4957,Z 124,A 2.6342,B 24.9457,C -1.7026,E1 25.1587,E2 443.3545} C_DIS
LIN {X 115.2354,Y 11.2303,Z 124,A 1.0594,B 24.9459,C -1.6998,E1 25.1592,E2 444.9266} C_DIS
LIN {X 115.5306,Y 7.5962,Z 124,A -0.7466,B 24.9462,C -1.6939,E1 25.1595,E2 446.7358} C_DIS
LIN {X 115.7223,Y 3.6499,Z 124,A -2.5973,B 24.9463,C -1.6925,E1 25.1597,E2 448.5789} C_DIS
LIN {X 115.7799,Y 0.4279,Z 124,A -4.225,B 24.9468,C -1.6857,E1 25.1597,E2 450.2129} C_DIS
LIN {X 115.7276,Y -3.4775,Z 124,A -6.1203,B 24.947,C -1.6811,E1 25.1597,E2 452.1076} C_DIS
LIN {X 115.5541,Y -7.2479,Z 124,A -8.0454,B 24.9476,C -1.6723,E1 25.1594,E2 454.042} C_DIS
LIN {X 115.2776,Y -10.7737,Z 124,A -9.7729,B 24.9479,C -1.6677,E1 25.159,E2 455.7703} C_DIS
LIN {X 114.9263,Y -14.0448,Z 124,A -11.2574,B 24.9478,C -1.6691,E1 25.1585,E2 457.2427} C_DIS
LIN {X 114.2506,Y -18.7586,Z 124,A -13.6924,B 24.9485,C -1.6577,E1 25.1575,E2 459.6901} C_DIS
LIN {X 113.7772,Y -21.4457,Z 124,A -15.8828,B 24.9512,C -1.6139,E1 25.1563,E2 461.9709} C_DIS
LIN {X 112.6034,Y -26.9389,Z 124,A -17.6261,B 24.9488,C -1.6535,E1 25.1553,E2 463.6107} C_DIS
LIN {X 111.6983,Y -30.4718,Z 124,A -19.5224,B 24.9494,C -1.6434,E1 25.1539,E2 465.52} C_DIS
LIN {X 110.7989,Y -33.6016,Z 124,A -21.2133,B 24.9499,C -1.6345,E1 25.1526,E2 467.2223} C_DIS
LIN {X 110.0457,Y -35.9867,Z 124,A -22.6506,B 24.9508,C -1.6212,E1 25.1513,E2 468.6827} C_DIS
LIN {X 108.4304,Y -40.5958,Z 124,A -24.7256,B 24.9502,C -1.6297,E1 25.1494,E2 470.7261} C_DIS
LIN {X 107.2739,Y -43.5578,Z 124,A -26.3377,B 24.9506,C -1.623,E1 25.1477,E2 472.3451} C_DIS
LIN {X 105.1658,Y -48.4287,Z 124,A -29.1212,B 24.9516,C -1.6075,E1 25.1445,E2 475.15} C_DIS
LIN {X 103.2659,Y -52.3571,Z 124,A -30.9029,B 24.9509,C -1.6187,E1 25.1424,E2 476.8956} C_DIS
LIN {X 101.9679,Y -54.8424,Z 124,A -32.5195,B 24.9518,C -1.6038,E1 25.1402,E2 478.539} C_DIS
LIN {X 100.3273,Y -57.7877,Z 124,A -34.4289,B 24.9528,C -1.5876,E1 25.1376,E2 480.4767} C_DIS
LIN {X 97.9841,Y -61.6785,Z 124,A -36.4825,B 24.9526,C -1.5901,E1 25.1346,E2 482.5138} C_DIS
LIN {X 95.4708,Y -65.504,Z 124,A -38.7676,B 24.9531,C -1.5828,E1 25.131,E2 484.805} C_DIS
LIN {X 93.2322,Y -68.65,Z 124,A -40.4757,B 24.9528,C -1.587,E1 25.1282,E2 486.4949} C_DIS
LIN {X 91.1226,Y -71.4272,Z 124,A -42.2814,B 24.9533,C -1.5785,E1 25.1251,E2 488.312} C_DIS
LIN {X 86.7174,Y -76.7172,Z 124,A -45.6175,B 24.9537,C -1.5728,E1 25.1192,E2 491.6464} C_DIS
LIN {X 83.8371,Y -79.8547,Z 124,A -47.7866,B 24.9541,C -1.5646,E1 25.115,E2 493.8253} C_DIS
LIN {X 81.8702,Y -81.8702,Z 124,A -49.8437,B 24.9561,C -1.5304,E1 25.1108,E2 495.9543} C_DIS
LIN {X 78.3844,Y -85.2107,Z 124,A -51.4482,B 24.9543,C -1.561,E1 25.1077,E2 497.4802} C_DIS
LIN {X 75.6901,Y -87.6147,Z 124,A -53.3189,B 24.9548,C -1.5529,E1 25.1037,E2 499.3626} C_DIS
LIN {X 72.3714,Y -90.3759,Z 124,A -55.6153,B 24.9555,C -1.5407,E1 25.0987,E2 501.6791} C_DIS
LIN {X 68.6619,Y -93.2235,Z 124,A -57.7307,B 24.9553,C -1.5449,E1 25.094,E2 503.7768} C_DIS
LIN {X 65.901,Y -95.1949,Z 124,A -59.423,B 24.9555,C -1.5409,E1 25.0901,E2 505.4729} C_DIS
LIN {X 62.6824,Y -97.3443,Z 124,A -61.241,B 24.9555,C -1.5415,E1 25.0859,E2 507.2833} C_DIS
LIN {X 57.4969,Y -100.4944,Z 124,A -64.2738,B 24.9559,C -1.5345,E1 25.0787,E2 510.3233} C_DIS
LIN {X 54.5377,Y -102.1325,Z 124,A -65.9615,B 24.9561,C -1.5309,E1 25.0745,E2 512.0147} C_DIS
LIN {X 51.0368,Y -103.925,Z 124,A -68.1492,B 24.9569,C -1.5167,E1 25.069,E2 514.2301} C_DIS
LIN {X 46.5587,Y -106.0064,Z 124,A -70.2493,B 24.9562,C -1.5285,E1 25.0637,E2 516.2969} C_DIS
LIN {X 43.6718,Y -107.2275,Z 124,A -71.6856,B 24.9561,C -1.5315,E1 25.06,E2 517.723} C_DIS
LIN {X 38.6022,Y -109.1555,Z 124,A -74.6552,B 24.957,C -1.5148,E1 25.0522,E2 520.7256} C_DIS
LIN {X 34.4474,Y -110.5368,Z 124,A -76.6517,B 24.9567,C -1.5199,E1 25.0469,E2 522.7064} C_DIS
LIN {X 30.1336,Y -111.7897,Z 124,A -79.392,B 24.9582,C -1.4942,E1 25.0394,E2 525.5029} C_DIS
LIN {X 26.4153,Y -112.7268,Z 124,A -81.0606,B 24.9577,C -1.5025,E1 25.0349,E2 527.1495} C_DIS
LIN {X 22.5274,Y -113.5689,Z 124,A -82.8713,B 24.9574,C -1.5078,E1 25.03,E2 528.9454} C_DIS
LIN {X 19.0325,Y -114.2048,Z 124,A -84.5434,B 24.9573,C -1.5103,E1 25.0254,E2 530.6098} C_DIS
LIN {X 15.859,Y -114.6894,Z 124,A -86.2192,B 24.9575,C -1.5053,E1 25.0208,E2 532.2959} C_DIS
LIN {X 12.3964,Y -115.1148,Z 124,A -87.6836,B 24.9569,C -1.5159,E1 25.0168,E2 533.7341} C_DIS
LIN {X 9.4473,Y -115.394,Z 124,A -89.3067,B 24.9574,C -1.5082,E1 25.0122,E2 535.3747} C_DIS
LIN {X 6.0936,Y -115.6197,Z 124,A -90.9571,B 24.9574,C -1.508,E1 25.0076,E2 537.0247} C_DIS
LIN {X 2.0868,Y -115.761,Z 124,A -93.0045,B 24.9576,C -1.5046,E1 25.0019,E2 539.0798} C_DIS
LIN {X 2.0868,Y -115.761,Z 124,A -93.0045,B 24.9576,C -1.5046,E1 25.0019,E2 539.0798} C_DIS
Enddeposition()
LIN {X 0.8107,Y -114.9091,Z 124,A -93.2846,B 24.9558,C -1.5352,E1 25.0013,E2 539.2873} C_DIS
Startdeposition()
$VEL.CP = VEL_PRINT
LIN {X 4.2214,Y -114.8365,Z 124,A -91.0359,B 24.9544,C -1.56,E1 25.0077,E2 536.9803} C_DIS
LIN {X 7.7705,Y -114.6489,Z 124,A -89.4168,B 24.9548,C -1.554,E1 25.0122,E2 535.3762} C_DIS
LIN {X 11.2623,Y -114.3609,Z 124,A -87.7018,B 24.9548,C -1.5534,E1 25.017,E2 533.6635} C_DIS
LIN {X 14.0602,Y -114.0507,Z 124,A -86.3002,B 24.9548,C -1.5542,E1 25.0209,E2 532.2611} C_DIS
LIN {X 16.8494,Y -113.672,Z 124,A -84.899,B 24.9547,C -1.5551,E1 25.0247,E2 530.859} C_DIS
LIN {X 19.0629,Y -113.3198,Z 124,A -83.7113,B 24.9545,C -1.5591,E1 25.028,E2 529.663} C_DIS
LIN {X 22.346,Y -112.72,Z 124,A -82.1219,B 24.9545,C -1.5571,E1 25.0324,E2 528.0801} C_DIS
LIN {X 24.7634,Y -112.2123,Z 124,A -80.8542,B 24.9545,C -1.5599,E1 25.0358,E2 526.8075} C_DIS
LIN {X 27.8816,Y -111.4801,Z 124,A -79.2995,B 24.9545,C -1.5595,E1 25.0401,E2 525.2559} C_DIS
LIN {X 30.4288,Y -110.811,Z 124,A -77.9973,B 24.9544,C -1.5605,E1 25.0436,E2 523.9536} C_DIS
LIN {X 33.285,Y -109.9875,Z 124,A -76.5106,B 24.9543,C -1.5624,E1 25.0476,E2 522.465} C_DIS
LIN {X 35.8127,Y -109.1898,Z 124,A -75.1773,B 24.9541,C -1.5645,E1 25.0511,E2 521.1291} C_DIS
LIN {X 38.6754,Y -108.21,Z 124,A -73.688,B 24.9541,C -1.5656,E1 25.055,E2 519.6402} C_DIS
LIN {X 41.2255,Y -107.2639,Z 124,A -72.3363,B 24.954,C -1.5673,E1 25.0586,E2 518.2875} C_DIS
LIN {X 43.4771,Y -106.3697,Z 124,A -71.0648,B 24.9537,C -1.5719,E1 25.0619,E2 517.0078} C_DIS
LIN {X 46.5619,Y -105.0582,Z 124,A -69.4654,B 24.9537,C -1.5711,E1 25.066,E2 515.4142} C_DIS
LIN {X 49.0541,Y -103.9174,Z 124,A -68.0962,B 24.9537,C -1.5734,E1 25.0694,E2 514.043} C_DIS
LIN {X 51.6045,Y -102.6749,Z 124,A -66.694,B 24.9535,C -1.5752,E1 25.0729,E2 512.6404} C_DIS
LIN {X 54.1623,Y -101.3493,Z 124,A -65.2627,B 24.9534,C -1.5774,E1 25.0765,E2 511.2079} C_DIS
LIN {X 56.6211,Y -99.9963,Z 124,A -63.8692,B 24.9532,C -1.5797,E1 25.0799,E2 509.8132} C_DIS
LIN {X 58.7778,Y -98.7423,Z 124,A -62.6022,B 24.953,C -1.5831,E1 25.0829,E2 508.542} C_DIS
LIN {X 61.3652,Y -97.1565,Z 124,A -61.1485,B 24.953,C -1.5832,E1 25.0864,E2 507.0926} C_DIS
LIN {X 63.8417,Y -95.5483,Z 124,A -59.6566,B 24.9528,C -1.587,E1 25.0899,E2 505.5966} C_DIS
LIN {X 66.1146,Y -93.9895,Z 124,A -58.2886,B 24.9527,C -1.5896,E1 25.093,E2 504.2272} C_DIS
LIN {X 68.3918,Y -92.3456,Z 124,A -56.8945,B 24.9525,C -1.5923,E1 25.0961,E2 502.8319} C_DIS
LIN {X 70.6865,Y -90.6016,Z 124,A -55.2804,B 24.9518,C -1.6036,E1 25.0998,E2 501.1968} C_DIS
LIN {X 73.4423,Y -88.3798,Z 124,A -53.708,B 24.9521,C -1.5986,E1 25.1031,E2 499.6421} C_DIS
LIN {X 75.586,Y -86.5535,Z 124,A -52.3082,B 24.9519,C -1.6017,E1 25.1061,E2 498.2407} C_DIS
LIN {X 77.6597,Y -84.6978,Z 124,A -50.9351,B 24.9518,C -1.6043,E1 25.1089,E2 496.8669} C_DIS
LIN {X 79.7007,Y -82.7802,Z 124,A -49.5432,B 24.9516,C -1.6075,E1 25.1117,E2 495.4733} C_DIS
LIN {X 81.7514,Y -80.7555,Z 124,A -48.1203,B 24.9514,C -1.6104,E1 25.1146,E2 494.0496} C_DIS
LIN {X 83.6799,Y -78.7555,Z 124,A -46.7302,B 24.9512,C -1.6141,E1 25.1172,E2 492.6567} C_DIS
LIN {X 85.5901,Y -76.6752,Z 124,A -45.3262,B 24.951,C -1.6175,E1 25.1199,E2 491.2508} C_DIS
LIN {X 87.4345,Y -74.5652,Z 124,A -43.9366,B 24.9508,C -1.6208,E1 25.1224,E2 489.8598} C_DIS
LIN {X 89.401,Y -72.196,Z 124,A -42.3577,B 24.9504,C -1.6269,E1 25.1252,E2 488.2737} C_DIS
LIN {X 91.2914,Y -69.7914,Z 124,A -40.8799,B 24.9503,C -1.6289,E1 25.1277,E2 486.7983} C_DIS
LIN {X 93.1321,Y -67.3177,Z 124,A -39.3719,B 24.9501,C -1.6317,E1 25.1302,E2 485.2909} C_DIS
LIN {X 94.75,Y -65.0205,Z 124,A -37.9794,B 24.9499,C -1.6352,E1 25.1324,E2 483.8968} C_DIS
LIN {X 96.2702,Y -62.7468,Z 124,A -36.6436,B 24.9497,C -1.6378,E1 25.1345,E2 482.5617} C_DIS
LIN {X 97.8353,Y -60.2784,Z 124,A -35.1779,B 24.9495,C -1.6424,E1 25.1367,E2 481.0925} C_DIS
LIN {X 99.2947,Y -57.8428,Z 124,A -33.7713,B 24.9492,C -1.6461,E1 25.1387,E2 479.6844} C_DIS
LIN {X 100.643,Y -55.4631,Z 124,A -32.4135,B 24.949,C -1.6499,E1 25.1405,E2 478.3248} C_DIS
LIN {X 101.9384,Y -53.0437,Z 124,A -31.0486,B 24.9487,C -1.6538,E1 25.1423,E2 476.9577} C_DIS
LIN {X 103.2664,Y -50.4112,Z 124,A -29.5935,B 24.9485,C -1.6576,E1 25.1441,E2 475.5016} C_DIS
LIN {X 104.4677,Y -47.8719,Z 124,A -28.2017,B 24.9483,C -1.6614,E1 25.1457,E2 474.1083} C_DIS
LIN {X 105.5764,Y -45.3732,Z 124,A -26.8623,B 24.9481,C -1.6645,E1 25.1472,E2 472.7689} C_DIS
LIN {X 106.6701,Y -42.7392,Z 124,A -25.4334,B 24.9478,C -1.6693,E1 25.1488,E2 471.3367} C_DIS
LIN {X 107.7116,Y -40.0432,Z 124,A -24.0035,B 24.9475,C -1.6732,E1 25.1502,E2 469.9054} C_DIS
LIN {X 108.6356,Y -37.4627,Z 124,A -22.6456,B 24.9473,C -1.6771,E1 25.1514,E2 468.546} C_DIS
LIN {X 109.5275,Y -34.769,Z 124,A -21.2393,B 24.947,C -1.6812,E1 25.1526,E2 467.138} C_DIS
LIN {X 110.3653,Y -32.0116,Z 124,A -19.8137,B 24.9468,C -1.6853,E1 25.1538,E2 465.7109} C_DIS
LIN {X 111.1144,Y -29.3057,Z 124,A -18.424,B 24.9465,C -1.6893,E1 25.1548,E2 464.3198} C_DIS
LIN {X 111.7858,Y -26.6286,Z 124,A -17.0552,B 24.9463,C -1.6934,E1 25.1557,E2 462.9493} C_DIS
LIN {X 112.3995,Y -23.9052,Z 124,A -15.6724,B 24.946,C -1.6975,E1 25.1565,E2 461.5649} C_DIS
LIN {X 112.9594,Y -21.1029,Z 124,A -14.2825,B 24.9458,C -1.7004,E1 25.1573,E2 460.1761} C_DIS
LIN {X 113.5605,Y -17.5716,Z 124,A -12.3754,B 24.9451,C -1.712,E1 25.1581,E2 458.2528} C_DIS
LIN {X 114.0501,Y -14.0654,Z 124,A -10.7331,B 24.9451,C -1.712,E1 25.1587,E2 456.6205} C_DIS
LIN {X 114.3527,Y -11.341,Z 124,A -9.4119,B 24.9449,C -1.7142,E1 25.1591,E2 455.3017} C_DIS
LIN {X 114.6613,Y -7.5867,Z 124,A -7.4493,B 24.9443,C -1.7244,E1 25.1595,E2 453.3268} C_DIS
LIN {X 114.8333,Y -4.2982,Z 124,A -5.877,B 24.9441,C -1.7264,E1 25.1597,E2 451.759} C_DIS
LIN {X 114.9041,Y -1.4841,Z 124,A -4.494,B 24.9439,C -1.7301,E1 25.1597,E2 450.3757} C_DIS
LIN {X 114.8906,Y 2.218,Z 124,A -2.6486,B 24.9435,C -1.7361,E1 25.1597,E2 448.5271} C_DIS
LIN {X 114.7994,Y 5.0869,Z 124,A -1.1597,B 24.943,C -1.7435,E1 25.1596,E2 447.0296} C_DIS
LIN {X 114.6075,Y 8.3825,Z 124,A 0.3853,B 24.943,C -1.744,E1 25.1593,E2 445.4925} C_DIS
LIN {X 114.3609,Y 11.2623,Z 124,A 1.8345,B 24.9427,C -1.749,E1 25.1589,E2 444.0401} C_DIS
LIN {X 114.0507,Y 14.0602,Z 124,A 3.2256,B 24.9424,C -1.7529,E1 25.1585,E2 442.6479} C_DIS
LIN {X 113.4655,Y 18.1859,Z 124,A 5.2941,B 24.942,C -1.7592,E1 25.1576,E2 440.577} C_DIS
LIN {X 112.986,Y 20.9598,Z 124,A 6.6861,B 24.9417,C -1.7631,E1 25.1569,E2 439.1839} C_DIS
LIN {X 112.4387,Y 23.7211,Z 124,A 8.0821,B 24.9415,C -1.7671,E1 25.1561,E2 437.7865} C_DIS
LIN {X 111.8172,Y 26.4968,Z 124,A 9.4893,B 24.9412,C -1.7711,E1 25.1553,E2 436.3782} C_DIS
LIN {X 111.1452,Y 29.1865,Z 124,A 10.8565,B 24.941,C -1.7746,E1 25.1543,E2 435.0104} C_DIS
LIN {X 110.4804,Y 31.6058,Z 124,A 12.0982,B 24.9407,C -1.7781,E1 25.1534,E2 433.7677} C_DIS
LIN {X 109.5726,Y 34.6264,Z 124,A 13.669,B 24.9404,C -1.7828,E1 25.1521,E2 432.1947} C_DIS
LIN {X 108.6629,Y 37.3848,Z 124,A 15.1054,B 24.9402,C -1.7866,E1 25.1508,E2 430.7574} C_DIS
LIN {X 107.7147,Y 40.0348,Z 124,A 16.6667,B 24.9394,C -1.7982,E1 25.1493,E2 429.1774} C_DIS
LIN {X 106.4268,Y 43.3369,Z 124,A 18.289,B 24.9394,C -1.7967,E1 25.1476,E2 427.5678} C_DIS
LIN {X 105.055,Y 46.5692,Z 124,A 19.9962,B 24.9393,C -1.7997,E1 25.1457,E2 425.8629} C_DIS
LIN {X 103.914,Y 49.0615,Z 124,A 21.3567,B 24.939,C -1.8033,E1 25.1441,E2 424.5011} C_DIS
LIN {X 102.6695,Y 51.6153,Z 124,A 22.7627,B 24.9388,C -1.8069,E1 25.1424,E2 423.0943} C_DIS
LIN {X 101.3462,Y 54.1683,Z 124,A 24.1883,B 24.9386,C -1.8105,E1 25.1405,E2 421.6677} C_DIS
LIN {X 99.9952,Y 56.6231,Z 124,A 25.5765,B 24.9383,C -1.8139,E1 25.1386,E2 420.2786} C_DIS
LIN {X 98.6236,Y 58.9787,Z 124,A 26.9085,B 24.9382,C -1.8163,E1 25.1367,E2 418.9478} C_DIS
LIN {X 97.3912,Y 60.9895,Z 124,A 28.1659,B 24.9377,C -1.8233,E1 25.1349,E2 417.6804} C_DIS
LIN {X 95.549,Y 63.8407,Z 124,A 29.7808,B 24.9377,C -1.824,E1 25.1324,E2 416.0717} C_DIS
LIN {X 93.9877,Y 66.1171,Z 124,A 31.1494,B 24.9374,C -1.8272,E1 25.1302,E2 414.7023} C_DIS
LIN {X 92.3425,Y 68.396,Z 124,A 32.5436,B 24.9372,C -1.8304,E1 25.1279,E2 413.3073} C_DIS
LIN {X 90.6193,Y 70.6636,Z 124,A 33.9566,B 24.937,C -1.8336,E1 25.1255,E2 411.8935} C_DIS
LIN {X 88.8639,Y 72.8587,Z 124,A 35.3504,B 24.9368,C -1.8366,E1 25.123,E2 410.499} C_DIS
LIN {X 86.7214,Y 75.3937,Z 124,A 37.0663,B 24.9363,C -1.8433,E1 25.1199,E2 408.7751} C_DIS
LIN {X 84.6905,Y 77.6677,Z 124,A 38.5093,B 24.9363,C -1.8433,E1 25.1172,E2 407.3387} C_DIS
LIN {X 82.7105,Y 79.773,Z 124,A 39.9921,B 24.936,C -1.8483,E1 25.1144,E2 405.8502} C_DIS
LIN {X 80.2542,Y 82.2467,Z 124,A 41.674,B 24.9359,C -1.8495,E1 25.111,E2 404.1728} C_DIS
LIN {X 78.2154,Y 84.1878,Z 124,A 43.0715,B 24.9357,C -1.8521,E1 25.1082,E2 402.7747} C_DIS
LIN {X 76.1574,Y 86.0537,Z 124,A 44.6272,B 24.935,C -1.8627,E1 25.1049,E2 401.2001} C_DIS
LIN {X 73.4279,Y 88.3917,Z 124,A 46.2342,B 24.9353,C -1.8578,E1 25.1015,E2 399.611} C_DIS
LIN {X 71.272,Y 90.1391,Z 124,A 47.6209,B 24.9351,C -1.8605,E1 25.0985,E2 398.2231} C_DIS
LIN {X 68.8061,Y 92.0355,Z 124,A 49.1836,B 24.9349,C -1.8639,E1 25.095,E2 396.6582} C_DIS
LIN {X 66.1742,Y 93.9479,Z 124,A 50.7748,B 24.9348,C -1.8652,E1 25.0914,E2 395.0693} C_DIS
LIN {X 64.1414,Y 95.3454,Z 124,A 52.0263,B 24.9346,C -1.8683,E1 25.0885,E2 393.8147} C_DIS
LIN {X 61.6608,Y 96.9688,Z 124,A 53.4476,B 24.9346,C -1.8681,E1 25.0852,E2 392.3986} C_DIS
LIN {X 59.1459,Y 98.5237,Z 124,A 54.9453,B 24.9344,C -1.8714,E1 25.0816,E2 390.8979} C_DIS
LIN {X 56.6425,Y 99.9844,Z 124,A 56.3834,B 24.9342,C -1.8731,E1 25.0781,E2 389.4599} C_DIS
LIN {X 54.2247,Y 101.3156,Z 124,A 57.7555,B 24.9342,C -1.8749,E1 25.0747,E2 388.0876} C_DIS
LIN {X 51.6732,Y 102.6407,Z 124,A 59.1852,B 24.934,C -1.8766,E1 25.0712,E2 386.6579} C_DIS
LIN {X 49.2226,Y 103.8376,Z 124,A 60.5432,B 24.9339,C -1.8782,E1 25.0678,E2 385.2996} C_DIS
LIN {X 46.6138,Y 105.0349,Z 124,A 61.9676,B 24.9338,C -1.8795,E1 25.0641,E2 383.8756} C_DIS
LIN {X 44.3561,Y 106.0065,Z 124,A 63.2271,B 24.9336,C -1.8824,E1 25.0609,E2 382.6122} C_DIS
LIN {X 41.3645,Y 107.2111,Z 124,A 64.7952,B 24.9336,C -1.8822,E1 25.0568,E2 381.0481} C_DIS
LIN {X 38.7793,Y 108.1727,Z 124,A 66.1689,B 24.9336,C -1.8834,E1 25.0532,E2 379.6744} C_DIS
LIN {X 36.1185,Y 109.0899,Z 124,A 67.5695,B 24.9334,C -1.8845,E1 25.0495,E2 378.2739} C_DIS
LIN {X 33.3655,Y 109.9636,Z 124,A 69.0073,B 24.9334,C -1.8855,E1 25.0457,E2 376.8363} C_DIS
LIN {X 30.6516,Y 110.7507,Z 124,A 70.4142,B 24.9333,C -1.8864,E1 25.0419,E2 375.4297} C_DIS
LIN {X 28.0073,Y 111.4483,Z 124,A 71.7759,B 24.9333,C -1.8872,E1 25.0382,E2 374.0682} C_DIS
LIN {X 25.5346,Y 112.0395,Z 124,A 73.067,B 24.9331,C -1.8889,E1 25.0347,E2 372.7747} C_DIS
LIN {X 22.5066,Y 112.688,Z 124,A 74.5828,B 24.9331,C -1.8884,E1 25.0306,E2 371.262} C_DIS
LIN {X 19.8929,Y 113.1779,Z 124,A 75.8805,B 24.9332,C -1.8877,E1 25.027,E2 369.9675} C_DIS
LIN {X 16.872,Y 113.6687,Z 124,A 77.434,B 24.9331,C -1.8893,E1 25.0227,E2 368.4116} C_DIS
LIN {X 13.1382,Y 114.1586,Z 124,A 79.3591,B 24.9329,C -1.8918,E1 25.0174,E2 366.482} C_DIS
LIN {X 9.9316,Y 114.4837,Z 124,A 80.9196,B 24.933,C -1.89,E1 25.0131,E2 364.927} C_DIS
LIN {X 7.4752,Y 114.6689,Z 124,A 82.1848,B 24.933,C -1.8916,E1 25.0095,E2 363.6584} C_DIS
LIN {X 4.2364,Y 114.8359,Z 124,A 83.9464,B 24.9325,C -1.8978,E1 25.0046,E2 361.8827} C_DIS
LIN {X 0.6907,Y 114.9099,Z 124,A 85.56,B 24.933,C -1.8908,E1 25.0001,E2 360.2858} C_DIS
LIN {X -2.8201,Y 114.8795,Z 124,A 87.2837,B 24.933,C -1.8892,E1 24.9953,E2 358.5658} C_DIS
LIN {X -5.6333,Y 114.7759,Z 124,A 88.6884,B 24.9331,C -1.8888,E1 24.9914,E2 357.1618} C_DIS
LIN {X -8.3691,Y 114.6084,Z 124,A 90.0429,B 24.9331,C -1.8877,E1 24.9876,E2 355.8094} C_DIS
LIN {X -10.8162,Y 114.402,Z 124,A 91.3311,B 24.9331,C -1.8899,E1 24.984,E2 354.5153} C_DIS
LIN {X -14.0654,Y 114.0501,Z 124,A 92.9136,B 24.9333,C -1.8869,E1 24.9796,E2 352.9389} C_DIS
LIN {X -16.8548,Y 113.6713,Z 124,A 94.319,B 24.9333,C -1.8861,E1 24.9758,E2 351.5343} C_DIS
LIN {X -19.6768,Y 113.2167,Z 124,A 95.7326,B 24.9334,C -1.8845,E1 24.9719,E2 350.1231} C_DIS
LIN {X -22.3502,Y 112.7192,Z 124,A 97.1046,B 24.9334,C -1.8841,E1 24.9681,E2 348.7505} C_DIS
LIN {X -25.1549,Y 112.1269,Z 124,A 98.5362,B 24.9335,C -1.883,E1 24.9642,E2 347.3199} C_DIS
LIN {X -27.8684,Y 111.4833,Z 124,A 99.9301,B 24.9336,C -1.8818,E1 24.9604,E2 345.9269} C_DIS
LIN {X -30.2046,Y 110.8715,Z 124,A 101.1806,B 24.9336,C -1.8825,E1 24.957,E2 344.6727} C_DIS
LIN {X -33.2669,Y 109.9929,Z 124,A 102.7237,B 24.9338,C -1.8788,E1 24.9529,E2 343.1359} C_DIS
LIN {X -36.0446,Y 109.1148,Z 124,A 104.1859,B 24.9339,C -1.8775,E1 24.949,E2 341.6742} C_DIS
LIN {X -38.7039,Y 108.2,Z 124,A 105.5916,B 24.934,C -1.8759,E1 24.9453,E2 340.2696} C_DIS
LIN {X -41.2704,Y 107.2468,Z 124,A 106.9394,B 24.9342,C -1.8733,E1 24.9418,E2 338.925} C_DIS
LIN {X -43.9492,Y 106.1776,Z 124,A 108.398,B 24.9342,C -1.8722,E1 24.9381,E2 337.4659} C_DIS
LIN {X -46.5639,Y 105.0573,Z 124,A 109.826,B 24.9344,C -1.8705,E1 24.9344,E2 336.0386} C_DIS
LIN {X -49.0776,Y 103.9065,Z 124,A 111.2147,B 24.9345,C -1.8688,E1 24.9309,E2 334.6504} C_DIS
LIN {X -51.6066,Y 102.6738,Z 124,A 112.6169,B 24.9347,C -1.8665,E1 24.9274,E2 333.2501} C_DIS
LIN {X -54.1706,Y 101.3449,Z 124,A 114.0617,B 24.9349,C -1.8642,E1 24.9238,E2 331.8066} C_DIS
LIN {X -56.6359,Y 99.9881,Z 124,A 115.4703,B 24.935,C -1.862,E1 24.9204,E2 330.3992} C_DIS
LIN {X -59.0033,Y 98.609,Z 124,A 116.8438,B 24.9352,C -1.8598,E1 24.9171,E2 329.0267} C_DIS
LIN {X -61.3995,Y 97.1351,Z 124,A 118.2512,B 24.9353,C -1.8574,E1 24.9138,E2 327.6207} C_DIS
LIN {X -63.8443,Y 95.5466,Z 124,A 119.7095,B 24.9355,C -1.8547,E1 24.9104,E2 326.164} C_DIS
LIN {X -66.095,Y 94.0031,Z 124,A 121.0767,B 24.9357,C -1.8522,E1 24.9072,E2 324.798} C_DIS
LIN {X -68.3662,Y 92.3643,Z 124,A 122.4792,B 24.9359,C -1.8496,E1 24.9041,E2 323.3968} C_DIS
LIN {X -71.1792,Y 90.2124,Z 124,A 124.2594,B 24.9361,C -1.8464,E1 24.9001,E2 321.6177} C_DIS
LIN {X -73.3997,Y 88.4152,Z 124,A 125.7004,B 24.9363,C -1.8439,E1 24.897,E2 320.1772} C_DIS
LIN {X -75.5948,Y 86.5458,Z 124,A 127.129,B 24.9365,C -1.8403,E1 24.894,E2 318.7516} C_DIS
LIN {X -77.6647,Y 84.6932,Z 124,A 128.5211,B 24.9367,C -1.8373,E1 24.8911,E2 317.3609} C_DIS
LIN {X -79.7159,Y 82.7655,Z 124,A 129.9319,B 24.9369,C -1.8343,E1 24.8883,E2 315.9516} C_DIS
LIN {X -81.7451,Y 80.7619,Z 124,A 131.3554,B 24.9372,C -1.8309,E1 24.8855,E2 314.5302} C_DIS
LIN {X -83.6886,Y 78.7462,Z 124,A 132.7651,B 24.9374,C -1.8279,E1 24.8828,E2 313.1213} C_DIS
LIN {X -85.5924,Y 76.6726,Z 124,A 134.185,B 24.9376,C -1.825,E1 24.8801,E2 311.7021} C_DIS
LIN {X -87.4449,Y 74.5529,Z 124,A 135.6116,B 24.9378,C -1.8223,E1 24.8775,E2 310.2755} C_DIS
LIN {X -89.2919,Y 72.3306,Z 124,A 137.0947,B 24.9378,C -1.8202,E1 24.8749,E2 308.7904} C_DIS
LIN {X -91.3978,Y 69.6532,Z 124,A 138.7458,B 24.9383,C -1.8137,E1 24.8721,E2 307.1471} C_DIS
LIN {X -93.039,Y 67.4447,Z 124,A 140.1206,B 24.9386,C -1.8101,E1 24.8698,E2 305.7743} C_DIS
LIN {X -94.4832,Y 65.4044,Z 124,A 141.4331,B 24.9386,C -1.8093,E1 24.8677,E2 304.4571} C_DIS
LIN {X -96.2855,Y 62.7236,Z 124,A 143.0019,B 24.9391,C -1.803,E1 24.8653,E2 302.8955} C_DIS
LIN {X -97.8291,Y 60.2885,Z 124,A 144.4467,B 24.9393,C -1.7992,E1 24.8632,E2 301.4524} C_DIS
LIN {X -99.2733,Y 57.8794,Z 124,A 145.8564,B 24.9396,C -1.7955,E1 24.8612,E2 300.0442} C_DIS
LIN {X -100.6215,Y 55.5015,Z 124,A 147.2278,B 24.9398,C -1.7918,E1 24.8593,E2 298.6743} C_DIS
LIN {X -101.8035,Y 53.2999,Z 124,A 148.5269,B 24.9399,C -1.7903,E1 24.8576,E2 297.372} C_DIS
LIN {X -103.2692,Y 50.4055,Z 124,A 150.1099,B 24.9403,C -1.784,E1 24.8556,E2 295.7954} C_DIS
LIN {X -104.4729,Y 47.8609,Z 124,A 151.5229,B 24.9406,C -1.7801,E1 24.854,E2 294.384} C_DIS
LIN {X -105.5841,Y 45.3555,Z 124,A 152.8985,B 24.9409,C -1.7763,E1 24.8524,E2 293.01} C_DIS
LIN {X -106.7055,Y 42.6517,Z 124,A 154.3652,B 24.9411,C -1.7721,E1 24.8509,E2 291.5452} C_DIS
LIN {X -107.7171,Y 40.0282,Z 124,A 155.7745,B 24.9414,C -1.768,E1 24.8495,E2 290.1376} C_DIS
LIN {X -108.6409,Y 37.4476,Z 124,A 157.1475,B 24.9417,C -1.764,E1 24.8482,E2 288.7665} C_DIS
LIN {X -109.5255,Y 34.7751,Z 124,A 158.5703,B 24.9419,C -1.7603,E1 24.847,E2 287.3442} C_DIS
LIN {X -110.3656,Y 32.0108,Z 124,A 160.019,B 24.9422,C -1.7561,E1 24.8459,E2 285.8972} C_DIS
LIN {X -111.1134,Y 29.3091,Z 124,A 161.4259,B 24.9425,C -1.752,E1 24.8448,E2 284.492} C_DIS
LIN {X -111.7865,Y 26.6255,Z 124,A 162.8228,B 24.9427,C -1.7483,E1 24.8439,E2 283.0958} C_DIS
LIN {X -112.4085,Y 23.8641,Z 124,A 164.2398,B 24.943,C -1.7439,E1 24.8431,E2 281.6808} C_DIS
LIN {X -112.9726,Y 21.0341,Z 124,A 165.6856,B 24.9433,C -1.7395,E1 24.8423,E2 280.2369} C_DIS
LIN {X -113.4412,Y 18.3364,Z 124,A 167.0621,B 24.9435,C -1.7356,E1 24.8417,E2 278.8616} C_DIS
LIN {X -113.8558,Y 15.5557,Z 124,A 168.4739,B 24.9438,C -1.7314,E1 24.8411,E2 277.4513} C_DIS
LIN {X -114.2021,Y 12.7668,Z 124,A 169.8829,B 24.9441,C -1.7272,E1 24.8407,E2 276.044} C_DIS
LIN {X -114.4763,Y 10.0113,Z 124,A 171.2797,B 24.9443,C -1.7233,E1 24.8403,E2 274.648} C_DIS
LIN {X -114.6956,Y 7.0803,Z 124,A 172.7484,B 24.9446,C -1.7187,E1 24.84,E2 273.1816} C_DIS
LIN {X -114.83,Y 4.3745,Z 124,A 174.112,B 24.9449,C -1.7148,E1 24.8399,E2 271.8191} C_DIS
LIN {X -114.9016,Y 1.6169,Z 124,A 175.4796,B 24.9452,C -1.71,E1 24.8398,E2 270.4546} C_DIS
LIN {X -114.9087,Y -0.9284,Z 124,A 176.8389,B 24.9452,C -1.7095,E1 24.8398,E2 269.0883} C_DIS
LIN {X -114.8413,Y -4.0659,Z 124,A 178.3757,B 24.9456,C -1.7033,E1 24.8399,E2 267.5571} C_DIS
LIN {X -114.6969,Y -7.0612,Z 124,A 179.848,B 24.946,C -1.6975,E1 24.8402,E2 266.0897} C_DIS
LIN {X -114.4996,Y -9.7442,Z 124,A -178.7933,B 24.9462,C -1.6939,E1 24.8405,E2 264.7315} C_DIS
LIN {X -114.2263,Y -12.5483,Z 124,A -177.3759,B 24.9465,C -1.6899,E1 24.8409,E2 263.3151} C_DIS
LIN {X -113.8792,Y -15.3843,Z 124,A -175.944,B 24.9468,C -1.6856,E1 24.8414,E2 261.8849} C_DIS
LIN {X -113.4701,Y -18.1566,Z 124,A -174.5369,B 24.947,C -1.6816,E1 24.842,E2 260.4791} C_DIS
LIN {X -112.9941,Y -20.9147,Z 124,A -173.1344,B 24.9473,C -1.6774,E1 24.8427,E2 259.078} C_DIS
LIN {X -112.4788,Y -23.5258,Z 124,A -171.7764,B 24.9475,C -1.6745,E1 24.8434,E2 257.719} C_DIS
LIN {X -111.8221,Y -26.4758,Z 124,A -170.2789,B 24.9478,C -1.6694,E1 24.8444,E2 256.2249} C_DIS
LIN {X -111.1226,Y -29.2745,Z 124,A -168.8329,B 24.948,C -1.6652,E1 24.8454,E2 254.7803} C_DIS
LIN {X -110.1254,Y -32.8204,Z 124,A -166.9183,B 24.9482,C -1.6628,E1 24.8468,E2 252.8605} C_DIS
LIN {X -109.1142,Y -36.0465,Z 124,A -165.2866,B 24.9486,C -1.6555,E1 24.8482,E2 251.237} C_DIS
LIN {X -108.1984,Y -38.7084,Z 124,A -163.8743,B 24.9489,C -1.6516,E1 24.8495,E2 249.8258} C_DIS
LIN {X -107.244,Y -41.2778,Z 124,A -162.5313,B 24.9492,C -1.6466,E1 24.8509,E2 248.4872} C_DIS
LIN {X -105.6111,Y -45.2937,Z 124,A -160.3253,B 24.9495,C -1.6421,E1 24.8532,E2 246.2797} C_DIS
LIN {X -104.5016,Y -47.7973,Z 124,A -158.9496,B 24.9497,C -1.6386,E1 24.8548,E2 244.9048} C_DIS
LIN {X -103.2684,Y -50.4071,Z 124,A -157.5034,B 24.9499,C -1.6348,E1 24.8566,E2 243.4598} C_DIS
LIN {X -102.1447,Y -52.6439,Z 124,A -156.2204,B 24.95,C -1.6327,E1 24.8582,E2 242.1748} C_DIS
LIN {X -100.6778,Y -55.4005,Z 124,A -154.6794,B 24.9504,C -1.6277,E1 24.8602,E2 240.6376} C_DIS
LIN {X -99.3287,Y -57.7835,Z 124,A -153.3295,B 24.9506,C -1.6234,E1 24.8621,E2 239.2909} C_DIS
LIN {X -97.895,Y -60.1802,Z 124,A -151.9034,B 24.9508,C -1.6211,E1 24.8642,E2 237.8631} C_DIS
LIN {X -96.358,Y -62.6123,Z 124,A -150.4582,B 24.951,C -1.6178,E1 24.8663,E2 236.4185} C_DIS
LIN {X -94.7958,Y -64.9532,Z 124,A -149.052,B 24.9512,C -1.6143,E1 24.8685,E2 235.0136} C_DIS
LIN {X -93.1766,Y -67.2553,Z 124,A -147.6411,B 24.9514,C -1.611,E1 24.8708,E2 233.6035} C_DIS
LIN {X -91.5015,Y -69.517,Z 124,A -146.2293,B 24.9516,C -1.6079,E1 24.8732,E2 232.1924} C_DIS
LIN {X -89.7258,Y -71.7949,Z 124,A -144.7826,B 24.9517,C -1.6047,E1 24.8757,E2 230.7465} C_DIS
LIN {X -87.9557,Y -73.9526,Z 124,A -143.3844,B 24.9519,C -1.6017,E1 24.8782,E2 229.349} C_DIS
LIN {X -86.1265,Y -76.0749,Z 124,A -141.9793,B 24.9521,C -1.5988,E1 24.8808,E2 227.9445} C_DIS
LIN {X -83.8498,Y -78.5749,Z 124,A -140.2506,B 24.9522,C -1.5968,E1 24.8841,E2 226.2129} C_DIS
LIN {X -81.7795,Y -80.7272,Z 124,A -138.7815,B 24.9525,C -1.5928,E1 24.8869,E2 224.7471} C_DIS
LIN {X -79.7767,Y -82.7069,Z 124,A -137.3798,B 24.9526,C -1.5897,E1 24.8897,E2 223.3469} C_DIS
LIN {X -77.7102,Y -84.6515,Z 124,A -135.9191,B 24.9527,C -1.5887,E1 24.8927,E2 221.8826} C_DIS
LIN {X -75.1003,Y -86.9777,Z 124,A -134.2076,B 24.953,C -1.5839,E1 24.8963,E2 220.1757} C_DIS
LIN {X -72.9654,Y -88.7761,Z 124,A -132.8101,B 24.9531,C -1.5815,E1 24.8993,E2 218.7787} C_DIS
LIN {X -70.6976,Y -90.5931,Z 124,A -131.3556,B 24.9533,C -1.579,E1 24.9025,E2 217.3246} C_DIS
LIN {X -68.4587,Y -92.2966,Z 124,A -129.947,B 24.9534,C -1.5768,E1 24.9056,E2 215.9163} C_DIS
LIN {X -66.1789,Y -93.9446,Z 124,A -128.5426,B 24.9536,C -1.5745,E1 24.9088,E2 214.5125} C_DIS
LIN {X -63.2727,Y -95.9235,Z 124,A -126.741,B 24.9536,C -1.5737,E1 24.913,E2 212.7068} C_DIS
LIN {X -60.2836,Y -97.8322,Z 124,A -125.0057,B 24.9538,C -1.5696,E1 24.9171,E2 210.9758} C_DIS
LIN {X -58.338,Y -99.0023,Z 124,A -123.797,B 24.9538,C -1.5712,E1 24.92,E2 209.7596} C_DIS
LIN {X -55.8004,Y -100.4546,Z 124,A -122.3659,B 24.9539,C -1.568,E1 24.9235,E2 208.3319} C_DIS
LIN {X -52.9997,Y -101.9616,Z 124,A -120.8156,B 24.9541,C -1.5644,E1 24.9273,E2 206.7859} C_DIS
LIN {X -50.4289,Y -103.2576,Z 124,A -119.3789,B 24.9542,C -1.5626,E1 24.9309,E2 205.3496} C_DIS
LIN {X -48.0328,Y -104.3928,Z 124,A -118.0859,B 24.9544,C -1.5599,E1 24.9342,E2 204.0599} C_DIS
LIN {X -45.3498,Y -105.5866,Z 124,A -116.585,B 24.9544,C -1.5599,E1 24.938,E2 202.5555} C_DIS
LIN {X -42.7322,Y -106.6729,Z 124,A -115.1661,B 24.9544,C -1.5587,E1 24.9417,E2 201.1363} C_DIS
LIN {X -40.0378,Y -107.7136,Z 124,A -113.7259,B 24.9546,C -1.5573,E1 24.9454,E2 199.6963} C_DIS
LIN {X -37.7672,Y -108.5287,Z 124,A -112.4864,B 24.9546,C -1.5579,E1 24.9487,E2 198.453} C_DIS
LIN {X -34.786,Y -109.522,Z 124,A -110.949,B 24.9546,C -1.5553,E1 24.9528,E2 196.9189} C_DIS
LIN {X -32.0155,Y -110.3642,Z 124,A -109.5052,B 24.9547,C -1.5543,E1 24.9566,E2 195.4751} C_DIS
LIN {X -29.3098,Y -111.1132,Z 124,A -108.1079,B 24.9547,C -1.5533,E1 24.9604,E2 194.0779} C_DIS
LIN {X -26.9875,Y -111.6982,Z 124,A -106.8586,B 24.9547,C -1.5551,E1 24.9638,E2 192.8227} C_DIS
LIN {X -23.8735,Y -112.4064,Z 124,A -105.3125,B 24.9549,C -1.5523,E1 24.968,E2 191.2812} C_DIS
LIN {X -21.0403,Y -112.9714,Z 124,A -103.8725,B 24.9549,C -1.5517,E1 24.972,E2 189.8411} C_DIS
LIN {X -17.5326,Y -113.5666,Z 124,A -102.0572,B 24.9549,C -1.553,E1 24.977,E2 188.021} C_DIS
LIN {X -14.0648,Y -114.0501,Z 124,A -100.3514,B 24.9549,C -1.5509,E1 24.9817,E2 186.319} C_DIS
LIN {X -11.3401,Y -114.3527,Z 124,A -98.9834,B 24.9549,C -1.5509,E1 24.9855,E2 184.9504} C_DIS
LIN {X -8.4616,Y -114.6021,Z 124,A -97.5428,B 24.9549,C -1.5508,E1 24.9895,E2 183.5093} C_DIS
LIN {X -5.7253,Y -114.7709,Z 124,A -96.1759,B 24.9549,C -1.5508,E1 24.9933,E2 182.1418} C_DIS
LIN {X -3.1358,Y -114.8698,Z 124,A -94.8631,B 24.9549,C -1.5519,E1 24.997,E2 180.8262} C_DIS
LIN {X -0.0029,Y -114.9141,Z 124,A -93.3227,B 24.9549,C -1.5513,E1 25.0013,E2 179.2873} C_DIS
LIN {X -0.0029,Y -114.9141,Z 124,A -93.3227,B 24.9549,C -1.5513,E1 25.0013,E2 179.2873} C_DIS
Enddeposition()
LIN {X 0.853,Y -120.6847,Z 125,A -93.0824,B 24.9606,C -1.4505,E1 25.0013,E2 179.286} C_DIS
Startdeposition()
$VEL.CP = VEL_PRINT
LIN {X -1.4811,Y -120.6809,Z 125,A -94.4582,B 24.9613,C -1.4377,E1 24.9974,E2 180.692} C_DIS
LIN {X -4.4423,Y -120.6082,Z 125,A -95.864,B 24.9613,C -1.4376,E1 24.9935,E2 182.0983} C_DIS
LIN {X -7.4008,Y -120.4629,Z 125,A -97.2702,B 24.9613,C -1.4375,E1 24.9895,E2 183.5052} C_DIS
LIN {X -10.3549,Y -120.2449,Z 125,A -98.6765,B 24.9613,C -1.4375,E1 24.9856,E2 184.912} C_DIS
LIN {X -13.3027,Y -119.9546,Z 125,A -100.083,B 24.9613,C -1.4376,E1 24.9817,E2 186.319} C_DIS
LIN {X -16.2425,Y -119.592,Z 125,A -101.4901,B 24.9613,C -1.4379,E1 24.9778,E2 187.7266} C_DIS
LIN {X -19.1726,Y -119.1574,Z 125,A -102.8969,B 24.9613,C -1.4382,E1 24.9739,E2 189.1338} C_DIS
LIN {X -23.0839,Y -118.4598,Z 125,A -104.8332,B 24.9613,C -1.4367,E1 24.9686,E2 191.0758} C_DIS
LIN {X -26.0888,Y -117.8348,Z 125,A -106.2739,B 24.9613,C -1.4381,E1 24.9647,E2 192.5149} C_DIS
LIN {X -29.3253,Y -117.0731,Z 125,A -107.8235,B 24.9611,C -1.4402,E1 24.9605,E2 194.0615} C_DIS
LIN {X -32.1896,Y -116.3181,Z 125,A -109.2315,B 24.9611,C -1.441,E1 24.9567,E2 195.4699} C_DIS
LIN {X -35.0345,Y -115.4931,Z 125,A -110.64,B 24.9611,C -1.4419,E1 24.9529,E2 196.8786} C_DIS
LIN {X -37.8582,Y -114.5985,Z 125,A -112.0488,B 24.961,C -1.4429,E1 24.9491,E2 198.2876} C_DIS
LIN {X -41.2603,Y -113.4157,Z 125,A -113.762,B 24.961,C -1.4443,E1 24.9446,E2 200.0008} C_DIS
LIN {X -44.0312,Y -112.369,Z 125,A -115.1711,B 24.9609,C -1.4455,E1 24.941,E2 201.4101} C_DIS
LIN {X -46.7756,Y -111.2545,Z 125,A -116.5805,B 24.9608,C -1.4468,E1 24.9373,E2 202.8195} C_DIS
LIN {X -49.4919,Y -110.0731,Z 125,A -118.0096,B 24.9608,C -1.4473,E1 24.9337,E2 204.2507} C_DIS
LIN {X -52.3599,Y -108.7381,Z 125,A -119.4959,B 24.9606,C -1.4498,E1 24.9299,E2 205.735} C_DIS
LIN {X -55.0127,Y -107.4204,Z 125,A -120.9057,B 24.9606,C -1.4514,E1 24.9264,E2 207.1447} C_DIS
LIN {X -57.6324,Y -106.0379,Z 125,A -122.3553,B 24.9606,C -1.4514,E1 24.9228,E2 208.5985} C_DIS
LIN {X -60.2173,Y -104.5916,Z 125,A -123.7265,B 24.9603,C -1.4549,E1 24.9195,E2 209.9653} C_DIS
LIN {X -62.9665,Y -102.9604,Z 125,A -125.2864,B 24.9603,C -1.4553,E1 24.9158,E2 211.5291} C_DIS
LIN {X -65.8153,Y -101.1653,Z 125,A -126.853,B 24.9601,C -1.4592,E1 24.9121,E2 213.0915} C_DIS
LIN {X -68.2782,Y -99.5197,Z 125,A -128.2642,B 24.96,C -1.4613,E1 24.9088,E2 214.5024} C_DIS
LIN {X -70.6999,Y -97.8141,Z 125,A -129.6754,B 24.9599,C -1.4635,E1 24.9056,E2 215.9133} C_DIS
LIN {X -73.9429,Y -95.3839,Z 125,A -131.6419,B 24.9598,C -1.4651,E1 24.9012,E2 217.8831} C_DIS
LIN {X -76.5649,Y -93.2946,Z 125,A -133.2047,B 24.9596,C -1.4693,E1 24.8979,E2 219.4417} C_DIS
LIN {X -78.8314,Y -91.3875,Z 125,A -134.6169,B 24.9594,C -1.4718,E1 24.8949,E2 220.8535} C_DIS
LIN {X -80.6455,Y -89.7879,Z 125,A -135.8329,B 24.9594,C -1.4711,E1 24.8923,E2 222.0759} C_DIS
LIN {X -83.2206,Y -87.4094,Z 125,A -137.4419,B 24.9591,C -1.4769,E1 24.889,E2 223.6776} C_DIS
LIN {X -85.2945,Y -85.3864,Z 125,A -138.8248,B 24.959,C -1.4795,E1 24.8863,E2 225.0601} C_DIS
LIN {X -87.4094,Y -83.2206,Z 125,A -140.2674,B 24.9588,C -1.4824,E1 24.8835,E2 226.502} C_DIS
LIN {X -89.4254,Y -81.0504,Z 125,A -141.6804,B 24.9587,C -1.4853,E1 24.8808,E2 227.9144} C_DIS
LIN {X -91.3875,Y -78.8314,Z 125,A -143.0933,B 24.9585,C -1.4883,E1 24.8782,E2 229.3267} C_DIS
LIN {X -93.2946,Y -76.5649,Z 125,A -144.5069,B 24.9583,C -1.4913,E1 24.8757,E2 230.7396} C_DIS
LIN {X -95.1455,Y -74.2523,Z 125,A -145.9205,B 24.9582,C -1.4944,E1 24.8733,E2 232.1526} C_DIS
LIN {X -96.9391,Y -71.8949,Z 125,A -147.3343,B 24.958,C -1.4975,E1 24.8709,E2 233.5656} C_DIS
LIN {X -98.6743,Y -69.4943,Z 125,A -148.7481,B 24.9578,C -1.5007,E1 24.8686,E2 234.9787} C_DIS
LIN {X -100.3501,Y -67.0518,Z 125,A -150.1621,B 24.9576,C -1.504,E1 24.8664,E2 236.3918} C_DIS
LIN {X -101.9654,Y -64.5689,Z 125,A -151.5764,B 24.9574,C -1.5074,E1 24.8643,E2 237.8053} C_DIS
LIN {X -103.5192,Y -62.047,Z 125,A -152.9908,B 24.9572,C -1.5108,E1 24.8622,E2 239.2188} C_DIS
LIN {X -104.8422,Y -59.7812,Z 125,A -154.2708,B 24.9572,C -1.5127,E1 24.8604,E2 240.501} C_DIS
LIN {X -106.4391,Y -56.8929,Z 125,A -155.8199,B 24.9568,C -1.5178,E1 24.8583,E2 242.0461} C_DIS
LIN {X -107.8032,Y -54.2636,Z 125,A -157.2345,B 24.9566,C -1.5214,E1 24.8566,E2 243.4598} C_DIS
LIN {X -109.1025,Y -51.6016,Z 125,A -158.6494,B 24.9564,C -1.525,E1 24.8548,E2 244.8737} C_DIS
LIN {X -110.336,Y -48.9086,Z 125,A -160.0645,B 24.9562,C -1.5287,E1 24.8532,E2 246.2878} C_DIS
LIN {X -111.503,Y -46.1861,Z 125,A -161.4795,B 24.956,C -1.5324,E1 24.8517,E2 247.7017} C_DIS
Enddeposition()
END
